LIN {X 0,Y 545.058,Z 281.586,A -85,B 0,C 180,E1 -3811.915,E2 -3811.915} C_VEL
LIN {X 0,Y 545.078,Z 281.584,A -85,B 0,C 180,E1 -3813.095,E2 -3813.095} C_VEL
LIN {X 0,Y 544.385,Z 281.672,A -85,B 0,C 180,E1 -3813.711,E2 -3813.711} C_VEL
LIN {X 0,Y 541.508,Z 282.03,A -85,B 0,C 180,E1 -3814.712,E2 -3814.712} C_VEL
LIN {X 0,Y 539.096,Z 282.331,A -85,B 0,C 180,E1 -3815.518,E2 -3815.518} C_VEL
LIN {X 0,Y 538.071,Z 282.462,A -85,B 0,C 180,E1 -3816.14,E2 -3816.14} C_VEL
LIN {X 0,Y 537.992,Z 282.467,A -85,B 0,C 180,E1 -3816.351,E2 -3816.351} C_VEL
LIN {X 0,Y 538.037,Z 282.462,A -85,B 0,C 180,E1 -3819.585,E2 -3819.585} C_VEL
LIN {X 0,Y 538.036,Z 282.468,A -85,B 0,C 180,E1 -3821.879,E2 -3821.879} C_VEL
LIN {X 0,Y 538.035,Z 282.461,A -85,B 0,C 180,E1 -3825.141,E2 -3825.141} C_VEL
LIN {X 0,Y 538.035,Z 282.463,A -85,B 0,C 180,E1 -3828.227,E2 -3828.227} C_VEL
LIN {X 0,Y 538.016,Z 282.466,A -85,B 0,C 180,E1 -3831.17,E2 -3831.17} C_VEL
LIN {X 0,Y 537.995,Z 282.469,A -85,B 0,C 180,E1 -3834.089,E2 -3834.089} C_VEL
LIN {X 0,Y 537.857,Z 282.645,A -85,B 0,C 180,E1 -3836.154,E2 -3836.154} C_VEL
LIN {X 0,Y 537.784,Z 288.557,A -85,B 0,C 180,E1 -3839.358,E2 -3839.358} C_VEL
LIN {X 0,Y 537.735,Z 293.055,A -85,B 0,C 180,E1 -3841.933,E2 -3841.933} C_VEL
LIN {X 0,Y 537.773,Z 297.369,A -85,B 0,C 180,E1 -3844.452,E2 -3844.452} C_VEL
LIN {X 0,Y 537.677,Z 301.678,A -85,B 0,C 180,E1 -3846.913,E2 -3846.913} C_VEL
LIN {X 0,Y 537.632,Z 305.956,A -85,B 0,C 180,E1 -3849.332,E2 -3849.332} C_VEL
LIN {X 0,Y 537.604,Z 310.176,A -85,B 0,C 180,E1 -3851.715,E2 -3851.715} C_VEL
LIN {X 0,Y 537.602,Z 314.303,A -85,B 0,C 180,E1 -3854.066,E2 -3854.066} C_VEL
LIN {X 0,Y 537.565,Z 318.7,A -85,B 0,C 180,E1 -3856.582,E2 -3856.582} C_VEL
LIN {X 0,Y 537.574,Z 318.943,A -85,B 0,C 180,E1 -3856.726,E2 -3856.726} C_VEL
LIN {X 0,Y 539.197,Z 329.347,A -85,B 0,C 180,E1 -3857.03,E2 -3857.03} C_VEL
LIN {X 0,Y 538.984,Z 342.462,A -85,B 0,C 180,E1 -3857.48,E2 -3857.48} C_VEL
LIN {X 0,Y 538.742,Z 354.682,A -85,B 0,C 180,E1 -3858.068,E2 -3858.068} C_VEL
LIN {X 0,Y 538.566,Z 365.025,A -85,B 0,C 180,E1 -3858.712,E2 -3858.712} C_VEL
LIN {X 0,Y 538.362,Z 374.875,A -85,B 0,C 180,E1 -3859.469,E2 -3859.469} C_VEL
LIN {X 0,Y 538.196,Z 383.038,A -85,B 0,C 180,E1 -3860.226,E2 -3860.226} C_VEL
LIN {X 0,Y 538.03,Z 389.945,A -85,B 0,C 180,E1 -3860.982,E2 -3860.982} C_VEL
LIN {X 0,Y 537.884,Z 395.929,A -85,B 0,C 180,E1 -3861.736,E2 -3861.736} C_VEL
LIN {X 0,Y 537.76,Z 402.268,A -85,B 0,C 180,E1 -3862.679,E2 -3862.679} C_VEL
LIN {X 0,Y 537.639,Z 407.848,A -85,B 0,C 180,E1 -3863.68,E2 -3863.68} C_VEL
LIN {X 0,Y 537.587,Z 412.691,A -85,B 0,C 180,E1 -3864.749,E2 -3864.749} C_VEL
LIN {X 0,Y 537.604,Z 416.69,A -85,B 0,C 180,E1 -3865.877,E2 -3865.877} C_VEL
LIN {X 0,Y 537.551,Z 419.653,A -85,B 0,C 180,E1 -3867.002,E2 -3867.002} C_VEL
LIN {X 0,Y 537.451,Z 422.149,A -85,B 0,C 180,E1 -3868.501,E2 -3868.501} C_VEL
LIN {X 0,Y 537.442,Z 422.734,A -85,B 0,C 180,E1 -3869.251,E2 -3869.251} C_VEL
LIN {X 0,Y 537.442,Z 422.804,A -85,B 0,C 180,E1 -3870.749,E2 -3870.749} C_VEL
LIN {X 0,Y 537.452,Z 422.221,A -85,B 0,C 180,E1 -3871.499,E2 -3871.499} C_VEL
LIN {X 0,Y 537.552,Z 419.867,A -85,B 0,C 180,E1 -3872.998,E2 -3872.998} C_VEL
LIN {X 0,Y 537.603,Z 416.98,A -85,B 0,C 180,E1 -3874.123,E2 -3874.123} C_VEL
LIN {X 0,Y 537.587,Z 413.06,A -85,B 0,C 180,E1 -3875.251,E2 -3875.251} C_VEL
LIN {X 0,Y 537.637,Z 408.312,A -85,B 0,C 180,E1 -3876.319,E2 -3876.319} C_VEL
LIN {X 0,Y 537.754,Z 402.817,A -85,B 0,C 180,E1 -3877.321,E2 -3877.321} C_VEL
LIN {X 0,Y 537.879,Z 396.581,A -85,B 0,C 180,E1 -3878.264,E2 -3878.264} C_VEL
LIN {X 0,Y 538.024,Z 389.105,A -85,B 0,C 180,E1 -3879.208,E2 -3879.208} C_VEL
LIN {X 0,Y 538.204,Z 382.044,A -85,B 0,C 180,E1 -3879.964,E2 -3879.964} C_VEL
LIN {X 0,Y 538.405,Z 373.693,A -85,B 0,C 180,E1 -3880.72,E2 -3880.72} C_VEL
LIN {X 0,Y 538.575,Z 363.07,A -85,B 0,C 180,E1 -3881.515,E2 -3881.515} C_VEL
LIN {X 0,Y 538.874,Z 350.602,A -85,B 0,C 180,E1 -3882.236,E2 -3882.236} C_VEL
LIN {X 0,Y 539.086,Z 338.621,A -85,B 0,C 180,E1 -3882.757,E2 -3882.757} C_VEL
LIN {X 0,Y 539.013,Z 326.997,A -85,B 0,C 180,E1 -3883.13,E2 -3883.13} C_VEL
LIN {X 0,Y 537.561,Z 318.988,A -85,B 0,C 180,E1 -3883.346,E2 -3883.346} C_VEL
LIN {X 0,Y 537.6,Z 314.46,A -85,B 0,C 180,E1 -3885.934,E2 -3885.934} C_VEL
LIN {X 0,Y 537.601,Z 310.355,A -85,B 0,C 180,E1 -3888.285,E2 -3888.285} C_VEL
LIN {X 0,Y 537.633,Z 306.122,A -85,B 0,C 180,E1 -3890.668,E2 -3890.668} C_VEL
LIN {X 0,Y 537.679,Z 301.842,A -85,B 0,C 180,E1 -3893.087,E2 -3893.087} C_VEL
LIN {X 0,Y 537.763,Z 297.422,A -85,B 0,C 180,E1 -3895.609,E2 -3895.609} C_VEL
LIN {X 0,Y 537.744,Z 291.815,A -85,B 0,C 180,E1 -3898.877,E2 -3898.877} C_VEL
LIN {X 0,Y 537.808,Z 286.54,A -85,B 0,C 180,E1 -3901.852,E2 -3901.852} C_VEL
LIN {X 0,Y 537.881,Z 282.489,A -85,B 0,C 180,E1 -3904.07,E2 -3904.07} C_VEL
LIN {X 0,Y 537.992,Z 282.474,A -85,B 0,C 180,E1 -3906.005,E2 -3906.005} C_VEL
LIN {X 0,Y 538.017,Z 282.469,A -85,B 0,C 180,E1 -3908.83,E2 -3908.83} C_VEL
LIN {X 0,Y 538.033,Z 282.466,A -85,B 0,C 180,E1 -3911.773,E2 -3911.773} C_VEL
LIN {X 0,Y 538.008,Z 282.472,A -85,B 0,C 180,E1 -3914.862,E2 -3914.862} C_VEL
LIN {X 0,Y 538.022,Z 282.468,A -85,B 0,C 180,E1 -3917.214,E2 -3917.214} C_VEL
LIN {X 0,Y 538.029,Z 282.47,A -85,B 0,C 180,E1 -3920.203,E2 -3920.203} C_VEL
LIN {X 0,Y 538.022,Z 282.468,A -85,B 0,C 180,E1 -3923.067,E2 -3923.067} C_VEL
LIN {X 0,Y 537.896,Z 282.486,A -85,B 0,C 180,E1 -3926.044,E2 -3926.044} C_VEL
LIN {X 0,Y 537.837,Z 282.622,A -85,B 0,C 180,E1 -3926.265,E2 -3926.265} C_VEL
LIN {X 0,Y 537.782,Z 288.721,A -85,B 0,C 180,E1 -3929.601,E2 -3929.601} C_VEL
LIN {X 0,Y 537.749,Z 294.411,A -85,B 0,C 180,E1 -3932.779,E2 -3932.779} C_VEL
LIN {X 0,Y 537.75,Z 298.878,A -85,B 0,C 180,E1 -3935.278,E2 -3935.278} C_VEL
LIN {X 0,Y 537.696,Z 304.615,A -85,B 0,C 180,E1 -3938.532,E2 -3938.532} C_VEL
LIN {X 0,Y 537.649,Z 308.817,A -85,B 0,C 180,E1 -3940.926,E2 -3940.926} C_VEL
LIN {X 0,Y 537.608,Z 313.006,A -85,B 0,C 180,E1 -3943.286,E2 -3943.286} C_VEL
LIN {X 0,Y 537.616,Z 316.936,A -85,B 0,C 180,E1 -3945.618,E2 -3945.618} C_VEL
LIN {X 0,Y 537.549,Z 318.912,A -85,B 0,C 180,E1 -3946.762,E2 -3946.762} C_VEL
LIN {X 0,Y 539.18,Z 328.814,A -85,B 0,C 180,E1 -3947.03,E2 -3947.03} C_VEL
LIN {X 0,Y 539.005,Z 342.142,A -85,B 0,C 180,E1 -3947.48,E2 -3947.48} C_VEL
LIN {X 0,Y 538.747,Z 353.631,A -85,B 0,C 180,E1 -3948.028,E2 -3948.028} C_VEL
LIN {X 0,Y 538.577,Z 363.06,A -85,B 0,C 180,E1 -3948.592,E2 -3948.592} C_VEL
LIN {X 0,Y 538.43,Z 371.298,A -85,B 0,C 180,E1 -3949.185,E2 -3949.185} C_VEL
LIN {X 0,Y 538.233,Z 379.087,A -85,B 0,C 180,E1 -3949.847,E2 -3949.847} C_VEL
LIN {X 0,Y 538.077,Z 386.623,A -85,B 0,C 180,E1 -3950.603,E2 -3950.603} C_VEL
LIN {X 0,Y 537.974,Z 393.094,A -85,B 0,C 180,E1 -3951.359,E2 -3951.359} C_VEL
LIN {X 0,Y 537.82,Z 399.898,A -85,B 0,C 180,E1 -3952.302,E2 -3952.302} C_VEL
LIN {X 0,Y 537.718,Z 405.583,A -85,B 0,C 180,E1 -3953.245,E2 -3953.245} C_VEL
LIN {X 0,Y 537.675,Z 411.113,A -85,B 0,C 180,E1 -3954.374,E2 -3954.374} C_VEL
LIN {X 0,Y 537.562,Z 415.464,A -85,B 0,C 180,E1 -3955.501,E2 -3955.501} C_VEL
LIN {X 0,Y 537.591,Z 417.825,A -85,B 0,C 180,E1 -3956.252,E2 -3956.252} C_VEL
LIN {X 0,Y 537.551,Z 419.682,A -85,B 0,C 180,E1 -3957.002,E2 -3957.002} C_VEL
LIN {X 0,Y 537.451,Z 422.122,A -85,B 0,C 180,E1 -3958.501,E2 -3958.501} C_VEL
LIN {X 0,Y 537.442,Z 422.755,A -85,B 0,C 180,E1 -3959.251,E2 -3959.251} C_VEL
LIN {X 0,Y 537.442,Z 422.786,A -85,B 0,C 180,E1 -3960.749,E2 -3960.749} C_VEL
LIN {X 0,Y 537.452,Z 422.232,A -85,B 0,C 180,E1 -3961.499,E2 -3961.499} C_VEL
LIN {X 0,Y 537.552,Z 419.859,A -85,B 0,C 180,E1 -3962.998,E2 -3962.998} C_VEL
LIN {X 0,Y 537.603,Z 416.977,A -85,B 0,C 180,E1 -3964.123,E2 -3964.123} C_VEL
LIN {X 0,Y 537.587,Z 413.06,A -85,B 0,C 180,E1 -3965.251,E2 -3965.251} C_VEL
LIN {X 0,Y 537.639,Z 408.305,A -85,B 0,C 180,E1 -3966.32,E2 -3966.32} C_VEL
LIN {X 0,Y 537.754,Z 402.819,A -85,B 0,C 180,E1 -3967.321,E2 -3967.321} C_VEL
LIN {X 0,Y 537.875,Z 396.582,A -85,B 0,C 180,E1 -3968.264,E2 -3968.264} C_VEL
LIN {X 0,Y 537.982,Z 390.729,A -85,B 0,C 180,E1 -3969.019,E2 -3969.019} C_VEL
LIN {X 0,Y 538.134,Z 383.935,A -85,B 0,C 180,E1 -3969.775,E2 -3969.775} C_VEL
LIN {X 0,Y 538.368,Z 374.742,A -85,B 0,C 180,E1 -3970.626,E2 -3970.626} C_VEL
LIN {X 0,Y 538.509,Z 366.147,A -85,B 0,C 180,E1 -3971.289,E2 -3971.289} C_VEL
LIN {X 0,Y 538.674,Z 356.599,A -85,B 0,C 180,E1 -3971.897,E2 -3971.897} C_VEL
LIN {X 0,Y 538.872,Z 346.258,A -85,B 0,C 180,E1 -3972.427,E2 -3972.427} C_VEL
LIN {X 0,Y 539.084,Z 335.494,A -85,B 0,C 180,E1 -3972.853,E2 -3972.853} C_VEL
LIN {X 0,Y 538.998,Z 327.101,A -85,B 0,C 180,E1 -3973.106,E2 -3973.106} C_VEL
LIN {X 0,Y 537.553,Z 319.061,A -85,B 0,C 180,E1 -3973.322,E2 -3973.322} C_VEL
LIN {X 0,Y 537.613,Z 314.728,A -85,B 0,C 180,E1 -3975.934,E2 -3975.934} C_VEL
LIN {X 0,Y 537.661,Z 309.18,A -85,B 0,C 180,E1 -3979.074,E2 -3979.074} C_VEL
LIN {X 0,Y 537.727,Z 304.116,A -85,B 0,C 180,E1 -3981.881,E2 -3981.881} C_VEL
LIN {X 0,Y 537.695,Z 298.715,A -85,B 0,C 180,E1 -3984.725,E2 -3984.725} C_VEL
LIN {X 0,Y 537.669,Z 293.664,A -85,B 0,C 180,E1 -3987.271,E2 -3987.271} C_VEL
LIN {X 0,Y 537.56,Z 288.115,A -85,B 0,C 180,E1 -3989.789,E2 -3989.789} C_VEL
LIN {X 0,Y 537.606,Z 282.523,A -85,B 0,C 180,E1 -3992.165,E2 -3992.165} C_VEL
LIN {X 0,Y 537.962,Z 282.477,A -85,B 0,C 180,E1 -3994.178,E2 -3994.178} C_VEL
LIN {X 0,Y 538.005,Z 282.47,A -85,B 0,C 180,E1 -3997.17,E2 -3997.17} C_VEL
LIN {X 0,Y 538.024,Z 282.467,A -85,B 0,C 180,E1 -3999.797,E2 -3999.797} C_VEL
LIN {X 0,Y 538.002,Z 282.471,A -85,B 0,C 180,E1 -4002.788,E2 -4002.788} C_VEL
LIN {X 0,Y 538.035,Z 282.466,A -85,B 0,C 180,E1 -4005.141,E2 -4005.141} C_VEL
LIN {X 0,Y 538.025,Z 282.469,A -85,B 0,C 180,E1 -4008.226,E2 -4008.226} C_VEL
LIN {X 0,Y 538.014,Z 282.472,A -85,B 0,C 180,E1 -4011.169,E2 -4011.169} C_VEL
LIN {X 0,Y 538.02,Z 282.572,A -85,B 0,C 180,E1 -4011.607,E2 -4011.607} C_VEL
LIN {X 0,Y 539.515,Z 290.583,A -85,B 0,C 180,E1 -4014.113,E2 -4014.113} C_VEL
LIN {X 0,Y 539.286,Z 299.975,A -85,B 0,C 180,E1 -4016.815,E2 -4016.815} C_VEL
LIN {X 0,Y 539.077,Z 309.293,A -85,B 0,C 180,E1 -4019.439,E2 -4019.439} C_VEL
LIN {X 0,Y 538.798,Z 320.333,A -85,B 0,C 180,E1 -4022.497,E2 -4022.497} C_VEL
LIN {X 0,Y 538.543,Z 330.78,A -85,B 0,C 180,E1 -4025.317,E2 -4025.317} C_VEL
LIN {X 0,Y 538.364,Z 340.735,A -85,B 0,C 180,E1 -4027.951,E2 -4027.951} C_VEL
LIN {X 0,Y 538.15,Z 352.266,A -85,B 0,C 180,E1 -4030.944,E2 -4030.944} C_VEL
LIN {X 0,Y 537.953,Z 363.009,A -85,B 0,C 180,E1 -4033.687,E2 -4033.687} C_VEL
LIN {X 0,Y 537.827,Z 374.712,A -85,B 0,C 180,E1 -4036.636,E2 -4036.636} C_VEL
LIN {X 0,Y 539.239,Z 384.519,A -85,B 0,C 180,E1 -4036.864,E2 -4036.864} C_VEL
LIN {X 0,Y 539.091,Z 397.175,A -85,B 0,C 180,E1 -4037.243,E2 -4037.243} C_VEL
LIN {X 0,Y 538.845,Z 409.485,A -85,B 0,C 180,E1 -4037.764,E2 -4037.764} C_VEL
LIN {X 0,Y 538.65,Z 420.458,A -85,B 0,C 180,E1 -4038.374,E2 -4038.374} C_VEL
LIN {X 0,Y 538.413,Z 431.925,A -85,B 0,C 180,E1 -4039.185,E2 -4039.185} C_VEL
LIN {X 0,Y 538.2,Z 441.6,A -85,B 0,C 180,E1 -4040.036,E2 -4040.036} C_VEL
LIN {X 0,Y 538.015,Z 450.412,A -85,B 0,C 180,E1 -4040.981,E2 -4040.981} C_VEL
LIN {X 0,Y 537.829,Z 459.001,A -85,B 0,C 180,E1 -4042.114,E2 -4042.114} C_VEL
LIN {X 0,Y 537.705,Z 465.868,A -85,B 0,C 180,E1 -4043.244,E2 -4043.244} C_VEL
LIN {X 0,Y 537.676,Z 471.366,A -85,B 0,C 180,E1 -4044.374,E2 -4044.374} C_VEL
LIN {X 0,Y 537.557,Z 475.677,A -85,B 0,C 180,E1 -4045.501,E2 -4045.501} C_VEL
LIN {X 0,Y 537.591,Z 477.957,A -85,B 0,C 180,E1 -4046.252,E2 -4046.252} C_VEL
LIN {X 0,Y 537.551,Z 479.808,A -85,B 0,C 180,E1 -4047.002,E2 -4047.002} C_VEL
LIN {X 0,Y 537.49,Z 481.198,A -85,B 0,C 180,E1 -4047.752,E2 -4047.752} C_VEL
LIN {X 0,Y 537.442,Z 482.785,A -85,B 0,C 180,E1 -4049.251,E2 -4049.251} C_VEL
LIN {X 0,Y 537.442,Z 483,A -85,B 0,C 180,E1 -4050,E2 -4050} C_VEL
LIN {X 0,Y 537.451,Z 482.186,A -85,B 0,C 180,E1 -4051.499,E2 -4051.499} C_VEL
LIN {X 0,Y 537.49,Z 481.199,A -85,B 0,C 180,E1 -4052.248,E2 -4052.248} C_VEL
LIN {X 0,Y 537.551,Z 479.81,A -85,B 0,C 180,E1 -4052.998,E2 -4052.998} C_VEL
LIN {X 0,Y 537.603,Z 476.896,A -85,B 0,C 180,E1 -4054.123,E2 -4054.123} C_VEL
LIN {X 0,Y 537.587,Z 472.949,A -85,B 0,C 180,E1 -4055.251,E2 -4055.251} C_VEL
LIN {X 0,Y 537.652,Z 468.087,A -85,B 0,C 180,E1 -4056.334,E2 -4056.334} C_VEL
LIN {X 0,Y 537.791,Z 461.468,A -85,B 0,C 180,E1 -4057.509,E2 -4057.509} C_VEL
LIN {X 0,Y 537.972,Z 453.478,A -85,B 0,C 180,E1 -4058.641,E2 -4058.641} C_VEL
LIN {X 0,Y 538.119,Z 445.335,A -85,B 0,C 180,E1 -4059.586,E2 -4059.586} C_VEL
LIN {X 0,Y 538.375,Z 435.4,A -85,B 0,C 180,E1 -4060.53,E2 -4060.53} C_VEL
LIN {X 0,Y 538.542,Z 425.586,A -85,B 0,C 180,E1 -4061.289,E2 -4061.289} C_VEL
LIN {X 0,Y 538.74,Z 414.594,A -85,B 0,C 180,E1 -4061.971,E2 -4061.971} C_VEL
LIN {X 0,Y 538.94,Z 402.108,A -85,B 0,C 180,E1 -4062.569,E2 -4062.569} C_VEL
LIN {X 0,Y 539.197,Z 389.087,A -85,B 0,C 180,E1 -4063.017,E2 -4063.017} C_VEL
LIN {X 0,Y 539.058,Z 382.364,A -85,B 0,C 180,E1 -4063.189,E2 -4063.189} C_VEL
LIN {X 0,Y 537.827,Z 374.712,A -85,B 0,C 180,E1 -4063.364,E2 -4063.364} C_VEL
LIN {X 0,Y 537.953,Z 363.009,A -85,B 0,C 180,E1 -4066.313,E2 -4066.313} C_VEL
LIN {X 0,Y 538.15,Z 352.266,A -85,B 0,C 180,E1 -4069.056,E2 -4069.056} C_VEL
LIN {X 0,Y 538.398,Z 339.988,A -85,B 0,C 180,E1 -4072.244,E2 -4072.244} C_VEL
LIN {X 0,Y 538.543,Z 330.78,A -85,B 0,C 180,E1 -4074.683,E2 -4074.683} C_VEL
LIN {X 0,Y 538.798,Z 320.333,A -85,B 0,C 180,E1 -4077.503,E2 -4077.503} C_VEL
LIN {X 0,Y 539.091,Z 309.026,A -85,B 0,C 180,E1 -4080.635,E2 -4080.635} C_VEL
LIN {X 0,Y 539.219,Z 299.631,A -85,B 0,C 180,E1 -4083.19,E2 -4083.19} C_VEL
LIN {X 0,Y 539.368,Z 291.385,A -85,B 0,C 180,E1 -4085.439,E2 -4085.439} C_VEL
LIN {X 0,Y 538.769,Z 286.486,A -85,B 0,C 180,E1 -4086.874,E2 -4086.874} C_VEL
LIN {X 0,Y 538.029,Z 282.469,A -85,B 0,C 180,E1 -4088.199,E2 -4088.199} C_VEL
LIN {X 0,Y 538.004,Z 282.473,A -85,B 0,C 180,E1 -4090.78,E2 -4090.78} C_VEL
LIN {X 0,Y 538.013,Z 282.468,A -85,B 0,C 180,E1 -4094.072,E2 -4094.072} C_VEL
LIN {X 0,Y 538,Z 282.469,A -85,B 0,C 180,E1 -4097.016,E2 -4097.016} C_VEL
LIN {X 0,Y 538.051,Z 282.461,A -85,B 0,C 180,E1 -4099.253,E2 -4099.253} C_VEL
LIN {X 0,Y 537.995,Z 282.474,A -85,B 0,C 180,E1 -4102.122,E2 -4102.122} C_VEL
LIN {X 0,Y 538.001,Z 282.467,A -85,B 0,C 180,E1 -4104.916,E2 -4104.916} C_VEL
LIN {X 0,Y 538.022,Z 282.47,A -85,B 0,C 180,E1 -4107.617,E2 -4107.617} C_VEL
LIN {X 0,Y 538.02,Z 282.467,A -85,B 0,C 180,E1 -4110.239,E2 -4110.239} C_VEL
LIN {X 0,Y 538.061,Z 282.461,A -85,B 0,C 180,E1 -4112.796,E2 -4112.796} C_VEL
LIN {X 0,Y 537.956,Z 282.479,A -85,B 0,C 180,E1 -4115.288,E2 -4115.288} C_VEL
LIN {X 0,Y 537.83,Z 282.494,A -85,B 0,C 180,E1 -4116.92,E2 -4116.92} C_VEL
LIN {X 0,Y 537.786,Z 283.612,A -85,B 0,C 180,E1 -4118.536,E2 -4118.536} C_VEL
LIN {X 0,Y 537.704,Z 285.905,A -85,B 0,C 180,E1 -4120.928,E2 -4120.928} C_VEL
LIN {X 0,Y 537.624,Z 287.92,A -85,B 0,C 180,E1 -4123.286,E2 -4123.286} C_VEL
LIN {X 0,Y 537.615,Z 289.979,A -85,B 0,C 180,E1 -4125.618,E2 -4125.618} C_VEL
LIN {X 0,Y 537.573,Z 291.236,A -85,B 0,C 180,E1 -4126.798,E2 -4126.798} C_VEL
LIN {X 0,Y 539.171,Z 300.777,A -85,B 0,C 180,E1 -4127.078,E2 -4127.078} C_VEL
LIN {X 0,Y 538.979,Z 312.274,A -85,B 0,C 180,E1 -4127.48,E2 -4127.48} C_VEL
LIN {X 0,Y 538.774,Z 322.521,A -85,B 0,C 180,E1 -4127.953,E2 -4127.953} C_VEL
LIN {X 0,Y 538.649,Z 331.507,A -85,B 0,C 180,E1 -4128.472,E2 -4128.472} C_VEL
LIN {X 0,Y 538.45,Z 340.354,A -85,B 0,C 180,E1 -4129.091,E2 -4129.091} C_VEL
LIN {X 0,Y 538.292,Z 348.295,A -85,B 0,C 180,E1 -4129.753,E2 -4129.753} C_VEL
LIN {X 0,Y 538.143,Z 355.087,A -85,B 0,C 180,E1 -4130.415,E2 -4130.415} C_VEL
LIN {X 0,Y 537.981,Z 361.742,A -85,B 0,C 180,E1 -4131.17,E2 -4131.17} C_VEL
LIN {X 0,Y 537.832,Z 368.713,A -85,B 0,C 180,E1 -4132.114,E2 -4132.114} C_VEL
LIN {X 0,Y 537.74,Z 374.517,A -85,B 0,C 180,E1 -4133.056,E2 -4133.056} C_VEL
LIN {X 0,Y 537.695,Z 379.406,A -85,B 0,C 180,E1 -4133.998,E2 -4133.998} C_VEL
LIN {X 0,Y 537.54,Z 384.136,A -85,B 0,C 180,E1 -4135.125,E2 -4135.125} C_VEL
LIN {X 0,Y 537.591,Z 387.77,A -85,B 0,C 180,E1 -4136.252,E2 -4136.252} C_VEL
LIN {X 0,Y 537.551,Z 389.661,A -85,B 0,C 180,E1 -4137.002,E2 -4137.002} C_VEL
LIN {X 0,Y 537.49,Z 391.132,A -85,B 0,C 180,E1 -4137.752,E2 -4137.752} C_VEL
LIN {X 0,Y 537.442,Z 392.717,A -85,B 0,C 180,E1 -4139.251,E2 -4139.251} C_VEL
LIN {X 0,Y 537.442,Z 392.996,A -85,B 0,C 180,E1 -4140,E2 -4140} C_VEL
LIN {X 0,Y 537.452,Z 392.187,A -85,B 0,C 180,E1 -4141.499,E2 -4141.499} C_VEL
LIN {X 0,Y 537.49,Z 391.282,A -85,B 0,C 180,E1 -4142.248,E2 -4142.248} C_VEL
LIN {X 0,Y 537.591,Z 388.019,A -85,B 0,C 180,E1 -4143.748,E2 -4143.748} C_VEL
LIN {X 0,Y 537.54,Z 384.465,A -85,B 0,C 180,E1 -4144.875,E2 -4144.875} C_VEL
LIN {X 0,Y 537.668,Z 379.815,A -85,B 0,C 180,E1 -4146.002,E2 -4146.002} C_VEL
LIN {X 0,Y 537.729,Z 373.953,A -85,B 0,C 180,E1 -4147.132,E2 -4147.132} C_VEL
LIN {X 0,Y 537.871,Z 366.768,A -85,B 0,C 180,E1 -4148.264,E2 -4148.264} C_VEL
LIN {X 0,Y 538.053,Z 357.614,A -85,B 0,C 180,E1 -4149.397,E2 -4149.397} C_VEL
LIN {X 0,Y 538.254,Z 349.208,A -85,B 0,C 180,E1 -4150.248,E2 -4150.248} C_VEL
LIN {X 0,Y 538.462,Z 340.199,A -85,B 0,C 180,E1 -4151.005,E2 -4151.005} C_VEL
LIN {X 0,Y 538.647,Z 330.368,A -85,B 0,C 180,E1 -4151.684,E2 -4151.684} C_VEL
LIN {X 0,Y 538.836,Z 320.495,A -85,B 0,C 180,E1 -4152.237,E2 -4152.237} C_VEL
LIN {X 0,Y 539.066,Z 308.575,A -85,B 0,C 180,E1 -4152.757,E2 -4152.757} C_VEL
LIN {X 0,Y 538.999,Z 298.562,A -85,B 0,C 180,E1 -4153.082,E2 -4153.082} C_VEL
LIN {X 0,Y 537.539,Z 290.625,A -85,B 0,C 180,E1 -4153.323,E2 -4153.323} C_VEL
LIN {X 0,Y 537.527,Z 287.909,A -85,B 0,C 180,E1 -4155.936,E2 -4155.936} C_VEL
LIN {X 0,Y 537.529,Z 285.425,A -85,B 0,C 180,E1 -4158.288,E2 -4158.288} C_VEL
LIN {X 0,Y 537.557,Z 282.839,A -85,B 0,C 180,E1 -4160.671,E2 -4160.671} C_VEL
LIN {X 0,Y 537.728,Z 282.507,A -85,B 0,C 180,E1 -4162.273,E2 -4162.273} C_VEL
LIN {X 0,Y 537.946,Z 282.48,A -85,B 0,C 180,E1 -4164.713,E2 -4164.713} C_VEL
LIN {X 0,Y 538.051,Z 282.458,A -85,B 0,C 180,E1 -4167.35,E2 -4167.35} C_VEL
LIN {X 0,Y 538.018,Z 282.463,A -85,B 0,C 180,E1 -4169.761,E2 -4169.761} C_VEL
LIN {X 0,Y 538.021,Z 282.469,A -85,B 0,C 180,E1 -4172.383,E2 -4172.383} C_VEL
LIN {X 0,Y 538.001,Z 282.464,A -85,B 0,C 180,E1 -4175.084,E2 -4175.084} C_VEL
LIN {X 0,Y 537.992,Z 282.467,A -85,B 0,C 180,E1 -4176.351,E2 -4176.351} C_VEL
LIN {X 0,Y 537.342,Z 282.55,A -85,B 0,C 180,E1 -4176.976,E2 -4176.976} C_VEL
LIN {X 0,Y 534.507,Z 282.907,A -85,B 0,C 180,E1 -4177.991,E2 -4177.991} C_VEL
LIN {X 0,Y 532.101,Z 283.202,A -85,B 0,C 180,E1 -4178.809,E2 -4178.809} C_VEL
LIN {X 0,Y 531.067,Z 283.33,A -85,B 0,C 180,E1 -4179.44,E2 -4179.44} C_VEL
LIN {X 0,Y 530.982,Z 283.342,A -85,B 0,C 180,E1 -4179.653,E2 -4179.653} C_VEL
LIN {X 0,Y 530.983,Z 283.343,A -85,B 0,C 180,E1 -4182.457,E2 -4182.457} C_VEL
LIN {X 0,Y 530.992,Z 283.343,A -85,B 0,C 180,E1 -4185.621,E2 -4185.621} C_VEL
LIN {X 0,Y 530.998,Z 283.338,A -85,B 0,C 180,E1 -4188.565,E2 -4188.565} C_VEL
LIN {X 0,Y 530.961,Z 283.349,A -85,B 0,C 180,E1 -4191.529,E2 -4191.529} C_VEL
LIN {X 0,Y 530.947,Z 283.346,A -85,B 0,C 180,E1 -4194.379,E2 -4194.379} C_VEL
LIN {X 0,Y 530.792,Z 283.494,A -85,B 0,C 180,E1 -4196.213,E2 -4196.213} C_VEL
LIN {X 0,Y 530.742,Z 288.452,A -85,B 0,C 180,E1 -4198.907,E2 -4198.907} C_VEL
LIN {X 0,Y 530.658,Z 293.031,A -85,B 0,C 180,E1 -4201.524,E2 -4201.524} C_VEL
LIN {X 0,Y 530.68,Z 297.632,A -85,B 0,C 180,E1 -4204.231,E2 -4204.231} C_VEL
LIN {X 0,Y 530.635,Z 301.709,A -85,B 0,C 180,E1 -4206.588,E2 -4206.588} C_VEL
LIN {X 0,Y 530.58,Z 306.024,A -85,B 0,C 180,E1 -4209.045,E2 -4209.045} C_VEL
LIN {X 0,Y 530.534,Z 310.312,A -85,B 0,C 180,E1 -4211.462,E2 -4211.462} C_VEL
LIN {X 0,Y 530.536,Z 314.532,A -85,B 0,C 180,E1 -4213.848,E2 -4213.848} C_VEL
LIN {X 0,Y 530.511,Z 319.204,A -85,B 0,C 180,E1 -4216.497,E2 -4216.497} C_VEL
LIN {X 0,Y 530.544,Z 319.671,A -85,B 0,C 180,E1 -4216.571,E2 -4216.571} C_VEL
LIN {X 0,Y 532.299,Z 329.735,A -85,B 0,C 180,E1 -4216.859,E2 -4216.859} C_VEL
LIN {X 0,Y 532.086,Z 342.841,A -85,B 0,C 180,E1 -4217.315,E2 -4217.315} C_VEL
LIN {X 0,Y 531.854,Z 354.465,A -85,B 0,C 180,E1 -4217.876,E2 -4217.876} C_VEL
LIN {X 0,Y 531.624,Z 365.46,A -85,B 0,C 180,E1 -4218.562,E2 -4218.562} C_VEL
LIN {X 0,Y 531.394,Z 376.467,A -85,B 0,C 180,E1 -4219.426,E2 -4219.426} C_VEL
LIN {X 0,Y 531.168,Z 385.371,A -85,B 0,C 180,E1 -4220.288,E2 -4220.288} C_VEL
LIN {X 0,Y 530.921,Z 394.959,A -85,B 0,C 180,E1 -4221.436,E2 -4221.436} C_VEL
LIN {X 0,Y 530.723,Z 402.633,A -85,B 0,C 180,E1 -4222.582,E2 -4222.582} C_VEL
LIN {X 0,Y 530.598,Z 408.624,A -85,B 0,C 180,E1 -4223.694,E2 -4223.694} C_VEL
LIN {X 0,Y 530.523,Z 412.913,A -85,B 0,C 180,E1 -4224.679,E2 -4224.679} C_VEL
LIN {X 0,Y 530.524,Z 416.848,A -85,B 0,C 180,E1 -4225.822,E2 -4225.822} C_VEL
LIN {X 0,Y 530.457,Z 419.771,A -85,B 0,C 180,E1 -4226.962,E2 -4226.962} C_VEL
LIN {X 0,Y 530.361,Z 422.226,A -85,B 0,C 180,E1 -4228.481,E2 -4228.481} C_VEL
LIN {X 0,Y 530.344,Z 422.815,A -85,B 0,C 180,E1 -4229.241,E2 -4229.241} C_VEL
LIN {X 0,Y 530.344,Z 422.874,A -85,B 0,C 180,E1 -4230.759,E2 -4230.759} C_VEL
LIN {X 0,Y 530.362,Z 422.308,A -85,B 0,C 180,E1 -4231.519,E2 -4231.519} C_VEL
LIN {X 0,Y 530.457,Z 419.975,A -85,B 0,C 180,E1 -4233.038,E2 -4233.038} C_VEL
LIN {X 0,Y 530.522,Z 417.13,A -85,B 0,C 180,E1 -4234.178,E2 -4234.178} C_VEL
LIN {X 0,Y 530.524,Z 413.272,A -85,B 0,C 180,E1 -4235.321,E2 -4235.321} C_VEL
LIN {X 0,Y 530.622,Z 407.604,A -85,B 0,C 180,E1 -4236.603,E2 -4236.603} C_VEL
LIN {X 0,Y 530.779,Z 400.832,A -85,B 0,C 180,E1 -4237.8,E2 -4237.8} C_VEL
LIN {X 0,Y 530.965,Z 392.736,A -85,B 0,C 180,E1 -4238.947,E2 -4238.947} C_VEL
LIN {X 0,Y 531.159,Z 384.396,A -85,B 0,C 180,E1 -4239.905,E2 -4239.905} C_VEL
LIN {X 0,Y 531.431,Z 374.14,A -85,B 0,C 180,E1 -4240.862,E2 -4240.862} C_VEL
LIN {X 0,Y 531.633,Z 363.877,A -85,B 0,C 180,E1 -4241.639,E2 -4241.639} C_VEL
LIN {X 0,Y 531.9,Z 352.842,A -85,B 0,C 180,E1 -4242.302,E2 -4242.302} C_VEL
LIN {X 0,Y 532.139,Z 340.239,A -85,B 0,C 180,E1 -4242.878,E2 -4242.878} C_VEL
LIN {X 0,Y 532.189,Z 328.249,A -85,B 0,C 180,E1 -4243.277,E2 -4243.277} C_VEL
LIN {X 0,Y 530.518,Z 319.32,A -85,B 0,C 180,E1 -4243.527,E2 -4243.527} C_VEL
LIN {X 0,Y 530.535,Z 314.703,A -85,B 0,C 180,E1 -4246.152,E2 -4246.152} C_VEL
LIN {X 0,Y 530.533,Z 310.484,A -85,B 0,C 180,E1 -4248.538,E2 -4248.538} C_VEL
LIN {X 0,Y 530.58,Z 306.191,A -85,B 0,C 180,E1 -4250.955,E2 -4250.955} C_VEL
LIN {X 0,Y 530.672,Z 300.899,A -85,B 0,C 180,E1 -4253.962,E2 -4253.962} C_VEL
LIN {X 0,Y 530.64,Z 296.104,A -85,B 0,C 180,E1 -4256.764,E2 -4256.764} C_VEL
LIN {X 0,Y 530.667,Z 291.696,A -85,B 0,C 180,E1 -4259.342,E2 -4259.342} C_VEL
LIN {X 0,Y 530.752,Z 286.867,A -85,B 0,C 180,E1 -4262.063,E2 -4262.063} C_VEL
LIN {X 0,Y 530.807,Z 283.37,A -85,B 0,C 180,E1 -4264.014,E2 -4264.014} C_VEL
LIN {X 0,Y 530.942,Z 283.351,A -85,B 0,C 180,E1 -4266.152,E2 -4266.152} C_VEL
LIN {X 0,Y 530.97,Z 283.348,A -85,B 0,C 180,E1 -4268.654,E2 -4268.654} C_VEL
LIN {X 0,Y 530.996,Z 283.343,A -85,B 0,C 180,E1 -4271.436,E2 -4271.436} C_VEL
LIN {X 0,Y 530.976,Z 283.346,A -85,B 0,C 180,E1 -4274.548,E2 -4274.548} C_VEL
LIN {X 0,Y 530.985,Z 283.345,A -85,B 0,C 180,E1 -4277.834,E2 -4277.834} C_VEL
LIN {X 0,Y 530.991,Z 283.343,A -85,B 0,C 180,E1 -4280.557,E2 -4280.557} C_VEL
LIN {X 0,Y 530.953,Z 283.348,A -85,B 0,C 180,E1 -4283.441,E2 -4283.441} C_VEL
LIN {X 0,Y 530.928,Z 283.352,A -85,B 0,C 180,E1 -4285.305,E2 -4285.305} C_VEL
LIN {X 0,Y 530.772,Z 283.442,A -85,B 0,C 180,E1 -4286.308,E2 -4286.308} C_VEL
LIN {X 0,Y 530.709,Z 289.065,A -85,B 0,C 180,E1 -4289.404,E2 -4289.404} C_VEL
LIN {X 0,Y 530.66,Z 294.691,A -85,B 0,C 180,E1 -4292.541,E2 -4292.541} C_VEL
LIN {X 0,Y 530.677,Z 298.921,A -85,B 0,C 180,E1 -4294.926,E2 -4294.926} C_VEL
LIN {X 0,Y 530.606,Z 304.337,A -85,B 0,C 180,E1 -4297.998,E2 -4297.998} C_VEL
LIN {X 0,Y 530.587,Z 308.987,A -85,B 0,C 180,E1 -4300.662,E2 -4300.662} C_VEL
LIN {X 0,Y 530.554,Z 313.208,A -85,B 0,C 180,E1 -4303.057,E2 -4303.057} C_VEL
LIN {X 0,Y 530.576,Z 317.205,A -85,B 0,C 180,E1 -4305.423,E2 -4305.423} C_VEL
LIN {X 0,Y 530.486,Z 319.187,A -85,B 0,C 180,E1 -4306.594,E2 -4306.594} C_VEL
LIN {X 0,Y 532.236,Z 329.509,A -85,B 0,C 180,E1 -4306.882,E2 -4306.882} C_VEL
LIN {X 0,Y 532.031,Z 343.207,A -85,B 0,C 180,E1 -4307.362,E2 -4307.362} C_VEL
LIN {X 0,Y 531.781,Z 354.258,A -85,B 0,C 180,E1 -4307.9,E2 -4307.9} C_VEL
LIN {X 0,Y 531.604,Z 363.383,A -85,B 0,C 180,E1 -4308.454,E2 -4308.454} C_VEL
LIN {X 0,Y 531.415,Z 372.652,A -85,B 0,C 180,E1 -4309.137,E2 -4309.137} C_VEL
LIN {X 0,Y 531.2,Z 381.287,A -85,B 0,C 180,E1 -4309.904,E2 -4309.904} C_VEL
LIN {X 0,Y 531.046,Z 388.551,A -85,B 0,C 180,E1 -4310.67,E2 -4310.67} C_VEL
LIN {X 0,Y 530.888,Z 394.76,A -85,B 0,C 180,E1 -4311.435,E2 -4311.435} C_VEL
LIN {X 0,Y 530.767,Z 401.315,A -85,B 0,C 180,E1 -4312.391,E2 -4312.391} C_VEL
LIN {X 0,Y 530.671,Z 405.796,A -85,B 0,C 180,E1 -4313.154,E2 -4313.154} C_VEL
LIN {X 0,Y 530.609,Z 411.288,A -85,B 0,C 180,E1 -4314.299,E2 -4314.299} C_VEL
LIN {X 0,Y 530.468,Z 415.607,A -85,B 0,C 180,E1 -4315.441,E2 -4315.441} C_VEL
LIN {X 0,Y 530.516,Z 417.944,A -85,B 0,C 180,E1 -4316.202,E2 -4316.202} C_VEL
LIN {X 0,Y 530.457,Z 419.779,A -85,B 0,C 180,E1 -4316.962,E2 -4316.962} C_VEL
LIN {X 0,Y 530.361,Z 422.199,A -85,B 0,C 180,E1 -4318.481,E2 -4318.481} C_VEL
LIN {X 0,Y 530.344,Z 422.824,A -85,B 0,C 180,E1 -4319.241,E2 -4319.241} C_VEL
LIN {X 0,Y 530.344,Z 422.858,A -85,B 0,C 180,E1 -4320.759,E2 -4320.759} C_VEL
LIN {X 0,Y 530.362,Z 422.311,A -85,B 0,C 180,E1 -4321.519,E2 -4321.519} C_VEL
LIN {X 0,Y 530.457,Z 419.964,A -85,B 0,C 180,E1 -4323.038,E2 -4323.038} C_VEL
LIN {X 0,Y 530.522,Z 417.112,A -85,B 0,C 180,E1 -4324.178,E2 -4324.178} C_VEL
LIN {X 0,Y 530.524,Z 413.239,A -85,B 0,C 180,E1 -4325.321,E2 -4325.321} C_VEL
LIN {X 0,Y 530.575,Z 409.017,A -85,B 0,C 180,E1 -4326.306,E2 -4326.306} C_VEL
LIN {X 0,Y 530.712,Z 403.076,A -85,B 0,C 180,E1 -4327.418,E2 -4327.418} C_VEL
LIN {X 0,Y 530.839,Z 396.869,A -85,B 0,C 180,E1 -4328.374,E2 -4328.374} C_VEL
LIN {X 0,Y 531.021,Z 389.388,A -85,B 0,C 180,E1 -4329.33,E2 -4329.33} C_VEL
LIN {X 0,Y 531.21,Z 382.258,A -85,B 0,C 180,E1 -4330.096,E2 -4330.096} C_VEL
LIN {X 0,Y 531.386,Z 373.801,A -85,B 0,C 180,E1 -4330.863,E2 -4330.863} C_VEL
LIN {X 0,Y 531.585,Z 364.802,A -85,B 0,C 180,E1 -4331.543,E2 -4331.543} C_VEL
LIN {X 0,Y 531.745,Z 355.836,A -85,B 0,C 180,E1 -4332.103,E2 -4332.103} C_VEL
LIN {X 0,Y 531.99,Z 344.14,A -85,B 0,C 180,E1 -4332.687,E2 -4332.687} C_VEL
LIN {X 0,Y 532.21,Z 330.754,A -85,B 0,C 180,E1 -4333.167,E2 -4333.167} C_VEL
LIN {X 0,Y 531.734,Z 326.201,A -85,B 0,C 180,E1 -4333.302,E2 -4333.302} C_VEL
LIN {X 0,Y 530.533,Z 319.568,A -85,B 0,C 180,E1 -4333.478,E2 -4333.478} C_VEL
LIN {X 0,Y 530.547,Z 315.062,A -85,B 0,C 180,E1 -4336.152,E2 -4336.152} C_VEL
LIN {X 0,Y 530.568,Z 310.862,A -85,B 0,C 180,E1 -4338.536,E2 -4338.536} C_VEL
LIN {X 0,Y 530.646,Z 306.498,A -85,B 0,C 180,E1 -4340.953,E2 -4340.953} C_VEL
LIN {X 0,Y 530.668,Z 300.849,A -85,B 0,C 180,E1 -4343.962,E2 -4343.962} C_VEL
LIN {X 0,Y 530.6,Z 295.325,A -85,B 0,C 180,E1 -4346.766,E2 -4346.766} C_VEL
LIN {X 0,Y 530.555,Z 289.702,A -85,B 0,C 180,E1 -4349.349,E2 -4349.349} C_VEL
LIN {X 0,Y 530.564,Z 283.401,A -85,B 0,C 180,E1 -4352.031,E2 -4352.031} C_VEL
LIN {X 0,Y 530.873,Z 283.362,A -85,B 0,C 180,E1 -4353.781,E2 -4353.781} C_VEL
LIN {X 0,Y 530.955,Z 283.351,A -85,B 0,C 180,E1 -4356.559,E2 -4356.559} C_VEL
LIN {X 0,Y 530.987,Z 283.344,A -85,B 0,C 180,E1 -4359.443,E2 -4359.443} C_VEL
LIN {X 0,Y 530.967,Z 283.346,A -85,B 0,C 180,E1 -4362.458,E2 -4362.458} C_VEL
LIN {X 0,Y 530.989,Z 283.345,A -85,B 0,C 180,E1 -4365.453,E2 -4365.453} C_VEL
LIN {X 0,Y 530.991,Z 283.345,A -85,B 0,C 180,E1 -4368.564,E2 -4368.564} C_VEL
LIN {X 0,Y 531,Z 283.466,A -85,B 0,C 180,E1 -4371.342,E2 -4371.342} C_VEL
LIN {X 0,Y 532.399,Z 290.726,A -85,B 0,C 180,E1 -4373.634,E2 -4373.634} C_VEL
LIN {X 0,Y 532.578,Z 294.949,A -85,B 0,C 180,E1 -4374.902,E2 -4374.902} C_VEL
LIN {X 0,Y 532.286,Z 304.562,A -85,B 0,C 180,E1 -4377.674,E2 -4377.674} C_VEL
LIN {X 0,Y 531.99,Z 315.432,A -85,B 0,C 180,E1 -4380.738,E2 -4380.738} C_VEL
LIN {X 0,Y 531.71,Z 326.114,A -85,B 0,C 180,E1 -4383.701,E2 -4383.701} C_VEL
LIN {X 0,Y 531.496,Z 336.919,A -85,B 0,C 180,E1 -4386.628,E2 -4386.628} C_VEL
LIN {X 0,Y 531.202,Z 349.197,A -85,B 0,C 180,E1 -4389.88,E2 -4389.88} C_VEL
LIN {X 0,Y 530.985,Z 361.475,A -85,B 0,C 180,E1 -4393.071,E2 -4393.071} C_VEL
LIN {X 0,Y 530.767,Z 374.52,A -85,B 0,C 180,E1 -4396.406,E2 -4396.406} C_VEL
LIN {X 0,Y 530.756,Z 374.712,A -85,B 0,C 180,E1 -4396.455,E2 -4396.455} C_VEL
LIN {X 0,Y 532.315,Z 385.435,A -85,B 0,C 180,E1 -4396.714,E2 -4396.714} C_VEL
LIN {X 0,Y 532.149,Z 398.473,A -85,B 0,C 180,E1 -4397.123,E2 -4397.123} C_VEL
LIN {X 0,Y 531.912,Z 409.486,A -85,B 0,C 180,E1 -4397.602,E2 -4397.602} C_VEL
LIN {X 0,Y 531.682,Z 421.021,A -85,B 0,C 180,E1 -4398.254,E2 -4398.254} C_VEL
LIN {X 0,Y 531.43,Z 431.924,A -85,B 0,C 180,E1 -4399.041,E2 -4399.041} C_VEL
LIN {X 0,Y 531.192,Z 441.6,A -85,B 0,C 180,E1 -4399.904,E2 -4399.904} C_VEL
LIN {X 0,Y 530.969,Z 450.412,A -85,B 0,C 180,E1 -4400.861,E2 -4400.861} C_VEL
LIN {X 0,Y 530.779,Z 459.002,A -85,B 0,C 180,E1 -4402.008,E2 -4402.008} C_VEL
LIN {X 0,Y 530.637,Z 465.868,A -85,B 0,C 180,E1 -4403.154,E2 -4403.154} C_VEL
LIN {X 0,Y 530.611,Z 471.366,A -85,B 0,C 180,E1 -4404.299,E2 -4404.299} C_VEL
LIN {X 0,Y 530.457,Z 475.677,A -85,B 0,C 180,E1 -4405.441,E2 -4405.441} C_VEL
LIN {X 0,Y 530.516,Z 477.957,A -85,B 0,C 180,E1 -4406.202,E2 -4406.202} C_VEL
LIN {X 0,Y 530.457,Z 479.808,A -85,B 0,C 180,E1 -4406.962,E2 -4406.962} C_VEL
LIN {X 0,Y 530.411,Z 481.197,A -85,B 0,C 180,E1 -4407.722,E2 -4407.722} C_VEL
LIN {X 0,Y 530.344,Z 482.785,A -85,B 0,C 180,E1 -4409.241,E2 -4409.241} C_VEL
LIN {X 0,Y 530.342,Z 483,A -85,B 0,C 180,E1 -4410,E2 -4410} C_VEL
LIN {X 0,Y 530.361,Z 482.186,A -85,B 0,C 180,E1 -4411.519,E2 -4411.519} C_VEL
LIN {X 0,Y 530.411,Z 481.199,A -85,B 0,C 180,E1 -4412.278,E2 -4412.278} C_VEL
LIN {X 0,Y 530.457,Z 479.81,A -85,B 0,C 180,E1 -4413.038,E2 -4413.038} C_VEL
LIN {X 0,Y 530.522,Z 476.896,A -85,B 0,C 180,E1 -4414.178,E2 -4414.178} C_VEL
LIN {X 0,Y 530.524,Z 472.949,A -85,B 0,C 180,E1 -4415.321,E2 -4415.321} C_VEL
LIN {X 0,Y 530.6,Z 467.261,A -85,B 0,C 180,E1 -4416.583,E2 -4416.583} C_VEL
LIN {X 0,Y 530.758,Z 460.237,A -85,B 0,C 180,E1 -4417.801,E2 -4417.801} C_VEL
LIN {X 0,Y 530.931,Z 451.99,A -85,B 0,C 180,E1 -4418.948,E2 -4418.948} C_VEL
LIN {X 0,Y 531.113,Z 443.538,A -85,B 0,C 180,E1 -4419.906,E2 -4419.906} C_VEL
LIN {X 0,Y 531.406,Z 433.097,A -85,B 0,C 180,E1 -4420.863,E2 -4420.863} C_VEL
LIN {X 0,Y 531.641,Z 421.313,A -85,B 0,C 180,E1 -4421.728,E2 -4421.728} C_VEL
LIN {X 0,Y 531.895,Z 409.485,A -85,B 0,C 180,E1 -4422.399,E2 -4422.399} C_VEL
LIN {X 0,Y 532.173,Z 397.168,A -85,B 0,C 180,E1 -4422.925,E2 -4422.925} C_VEL
LIN {X 0,Y 532.284,Z 384.034,A -85,B 0,C 180,E1 -4423.323,E2 -4423.323} C_VEL
LIN {X 0,Y 530.756,Z 374.712,A -85,B 0,C 180,E1 -4423.545,E2 -4423.545} C_VEL
LIN {X 0,Y 530.939,Z 363.009,A -85,B 0,C 180,E1 -4426.535,E2 -4426.535} C_VEL
LIN {X 0,Y 531.139,Z 352.266,A -85,B 0,C 180,E1 -4429.317,E2 -4429.317} C_VEL
LIN {X 0,Y 531.376,Z 341.29,A -85,B 0,C 180,E1 -4432.207,E2 -4432.207} C_VEL
LIN {X 0,Y 531.564,Z 332.314,A -85,B 0,C 180,E1 -4434.612,E2 -4434.612} C_VEL
LIN {X 0,Y 531.827,Z 321.033,A -85,B 0,C 180,E1 -4437.7,E2 -4437.7} C_VEL
LIN {X 0,Y 532.122,Z 311.049,A -85,B 0,C 180,E1 -4440.487,E2 -4440.487} C_VEL
LIN {X 0,Y 532.221,Z 300.765,A -85,B 0,C 180,E1 -4443.231,E2 -4443.231} C_VEL
LIN {X 0,Y 532.406,Z 292.563,A -85,B 0,C 180,E1 -4445.508,E2 -4445.508} C_VEL
LIN {X 0,Y 531.785,Z 287.738,A -85,B 0,C 180,E1 -4446.965,E2 -4446.965} C_VEL
LIN {X 0,Y 530.965,Z 283.35,A -85,B 0,C 180,E1 -4448.41,E2 -4448.41} C_VEL
LIN {X 0,Y 530.964,Z 283.347,A -85,B 0,C 180,E1 -4451.439,E2 -4451.439} C_VEL
LIN {X 0,Y 530.97,Z 283.349,A -85,B 0,C 180,E1 -4454.549,E2 -4454.549} C_VEL
LIN {X 0,Y 530.974,Z 283.344,A -85,B 0,C 180,E1 -4457.836,E2 -4457.836} C_VEL
LIN {X 0,Y 530.991,Z 283.345,A -85,B 0,C 180,E1 -4460.557,E2 -4460.557} C_VEL
LIN {X 0,Y 530.958,Z 283.346,A -85,B 0,C 180,E1 -4463.442,E2 -4463.442} C_VEL
LIN {X 0,Y 531.002,Z 283.341,A -85,B 0,C 180,E1 -4466.494,E2 -4466.494} C_VEL
LIN {X 0,Y 530.977,Z 283.346,A -85,B 0,C 180,E1 -4469.355,E2 -4469.355} C_VEL
LIN {X 0,Y 531.016,Z 283.338,A -85,B 0,C 180,E1 -4472.468,E2 -4472.468} C_VEL
LIN {X 0,Y 530.943,Z 283.351,A -85,B 0,C 180,E1 -4474.939,E2 -4474.939} C_VEL
LIN {X 0,Y 530.739,Z 283.556,A -85,B 0,C 180,E1 -4477.417,E2 -4477.417} C_VEL
LIN {X 0,Y 530.745,Z 285.992,A -85,B 0,C 180,E1 -4480.08,E2 -4480.08} C_VEL
LIN {X 0,Y 530.625,Z 288.697,A -85,B 0,C 180,E1 -4483.059,E2 -4483.059} C_VEL
LIN {X 0,Y 530.608,Z 290.771,A -85,B 0,C 180,E1 -4485.424,E2 -4485.424} C_VEL
LIN {X 0,Y 530.529,Z 291.924,A -85,B 0,C 180,E1 -4486.632,E2 -4486.632} C_VEL
LIN {X 0,Y 532.248,Z 301.676,A -85,B 0,C 180,E1 -4486.931,E2 -4486.931} C_VEL
LIN {X 0,Y 532.026,Z 313.693,A -85,B 0,C 180,E1 -4487.362,E2 -4487.362} C_VEL
LIN {X 0,Y 531.854,Z 324.393,A -85,B 0,C 180,E1 -4487.874,E2 -4487.874} C_VEL
LIN {X 0,Y 531.644,Z 335.67,A -85,B 0,C 180,E1 -4488.563,E2 -4488.563} C_VEL
LIN {X 0,Y 531.395,Z 346.767,A -85,B 0,C 180,E1 -4489.426,E2 -4489.426} C_VEL
LIN {X 0,Y 531.166,Z 355.675,A -85,B 0,C 180,E1 -4490.288,E2 -4490.288} C_VEL
LIN {X 0,Y 530.975,Z 363.825,A -85,B 0,C 180,E1 -4491.245,E2 -4491.245} C_VEL
LIN {X 0,Y 530.823,Z 370.592,A -85,B 0,C 180,E1 -4492.2,E2 -4492.2} C_VEL
LIN {X 0,Y 530.703,Z 376.213,A -85,B 0,C 180,E1 -4493.155,E2 -4493.155} C_VEL
LIN {X 0,Y 530.647,Z 380.018,A -85,B 0,C 180,E1 -4493.918,E2 -4493.918} C_VEL
LIN {X 0,Y 530.504,Z 384.676,A -85,B 0,C 180,E1 -4495.06,E2 -4495.06} C_VEL
LIN {X 0,Y 530.516,Z 388.237,A -85,B 0,C 180,E1 -4496.202,E2 -4496.202} C_VEL
LIN {X 0,Y 530.486,Z 390.094,A -85,B 0,C 180,E1 -4496.962,E2 -4496.962} C_VEL
LIN {X 0,Y 530.412,Z 391.538,A -85,B 0,C 180,E1 -4497.722,E2 -4497.722} C_VEL
LIN {X 0,Y 530.353,Z 393.091,A -85,B 0,C 180,E1 -4499.241,E2 -4499.241} C_VEL
LIN {X 0,Y 530.352,Z 393.359,A -85,B 0,C 180,E1 -4500,E2 -4500} C_VEL
LIN {X 0,Y 530.363,Z 392.554,A -85,B 0,C 180,E1 -4501.519,E2 -4501.519} C_VEL
LIN {X 0,Y 530.412,Z 391.655,A -85,B 0,C 180,E1 -4502.278,E2 -4502.278} C_VEL
LIN {X 0,Y 530.516,Z 388.433,A -85,B 0,C 180,E1 -4503.798,E2 -4503.798} C_VEL
LIN {X 0,Y 530.485,Z 384.931,A -85,B 0,C 180,E1 -4504.94,E2 -4504.94} C_VEL
LIN {X 0,Y 530.607,Z 380.329,A -85,B 0,C 180,E1 -4506.083,E2 -4506.083} C_VEL
LIN {X 0,Y 530.696,Z 374.518,A -85,B 0,C 180,E1 -4507.228,E2 -4507.228} C_VEL
LIN {X 0,Y 530.87,Z 367.277,A -85,B 0,C 180,E1 -4508.374,E2 -4508.374} C_VEL
LIN {X 0,Y 531.059,Z 358.076,A -85,B 0,C 180,E1 -4509.522,E2 -4509.522} C_VEL
LIN {X 0,Y 531.289,Z 349.629,A -85,B 0,C 180,E1 -4510.383,E2 -4510.383} C_VEL
LIN {X 0,Y 531.495,Z 340.577,A -85,B 0,C 180,E1 -4511.151,E2 -4511.151} C_VEL
LIN {X 0,Y 531.698,Z 331.267,A -85,B 0,C 180,E1 -4511.802,E2 -4511.802} C_VEL
LIN {X 0,Y 531.912,Z 320.763,A -85,B 0,C 180,E1 -4512.398,E2 -4512.398} C_VEL
LIN {X 0,Y 532.137,Z 308.707,A -85,B 0,C 180,E1 -4512.926,E2 -4512.926} C_VEL
LIN {X 0,Y 532.089,Z 299.812,A -85,B 0,C 180,E1 -4513.219,E2 -4513.219} C_VEL
LIN {X 0,Y 530.475,Z 291.192,A -85,B 0,C 180,E1 -4513.479,E2 -4513.479} C_VEL
LIN {X 0,Y 530.473,Z 288.338,A -85,B 0,C 180,E1 -4516.154,E2 -4516.154} C_VEL
LIN {X 0,Y 530.458,Z 285.768,A -85,B 0,C 180,E1 -4518.541,E2 -4518.541} C_VEL
LIN {X 0,Y 530.518,Z 283.405,A -85,B 0,C 180,E1 -4520.958,E2 -4520.958} C_VEL
LIN {X 0,Y 530.771,Z 283.372,A -85,B 0,C 180,E1 -4523.405,E2 -4523.405} C_VEL
LIN {X 0,Y 530.977,Z 283.339,A -85,B 0,C 180,E1 -4525.899,E2 -4525.899} C_VEL
LIN {X 0,Y 530.991,Z 283.344,A -85,B 0,C 180,E1 -4528.456,E2 -4528.456} C_VEL
LIN {X 0,Y 530.957,Z 283.342,A -85,B 0,C 180,E1 -4531.079,E2 -4531.079} C_VEL
LIN {X 0,Y 530.99,Z 283.34,A -85,B 0,C 180,E1 -4533.773,E2 -4533.773} C_VEL
LIN {X 0,Y 530.958,Z 283.348,A -85,B 0,C 180,E1 -4536.558,E2 -4536.558} C_VEL
LIN {X 0,Y 530.982,Z 283.342,A -85,B 0,C 180,E1 -4539.653,E2 -4539.653} C_VEL
LIN {X 0,Y 530.311,Z 283.431,A -85,B 0,C 180,E1 -4540.286,E2 -4540.286} C_VEL
LIN {X 0,Y 527.446,Z 283.786,A -85,B 0,C 180,E1 -4541.313,E2 -4541.313} C_VEL
LIN {X 0,Y 525.031,Z 284.089,A -85,B 0,C 180,E1 -4542.141,E2 -4542.141} C_VEL
LIN {X 0,Y 524.001,Z 284.211,A -85,B 0,C 180,E1 -4542.78,E2 -4542.78} C_VEL
LIN {X 0,Y 523.921,Z 284.22,A -85,B 0,C 180,E1 -4542.996,E2 -4542.996} C_VEL
LIN {X 0,Y 523.945,Z 284.223,A -85,B 0,C 180,E1 -4545.772,E2 -4545.772} C_VEL
LIN {X 0,Y 523.943,Z 284.216,A -85,B 0,C 180,E1 -4548.908,E2 -4548.908} C_VEL
LIN {X 0,Y 523.919,Z 284.225,A -85,B 0,C 180,E1 -4551.898,E2 -4551.898} C_VEL
LIN {X 0,Y 523.875,Z 284.228,A -85,B 0,C 180,E1 -4554.919,E2 -4554.919} C_VEL
LIN {X 0,Y 523.736,Z 284.402,A -85,B 0,C 180,E1 -4556.303,E2 -4556.303} C_VEL
LIN {X 0,Y 523.66,Z 289.906,A -85,B 0,C 180,E1 -4559.336,E2 -4559.336} C_VEL
LIN {X 0,Y 523.609,Z 295.124,A -85,B 0,C 180,E1 -4562.359,E2 -4562.359} C_VEL
LIN {X 0,Y 523.583,Z 300.283,A -85,B 0,C 180,E1 -4565.411,E2 -4565.411} C_VEL
LIN {X 0,Y 523.528,Z 304.614,A -85,B 0,C 180,E1 -4567.921,E2 -4567.921} C_VEL
LIN {X 0,Y 523.503,Z 308.97,A -85,B 0,C 180,E1 -4570.389,E2 -4570.389} C_VEL
LIN {X 0,Y 523.478,Z 313.308,A -85,B 0,C 180,E1 -4572.821,E2 -4572.821} C_VEL
LIN {X 0,Y 523.512,Z 317.584,A -85,B 0,C 180,E1 -4575.222,E2 -4575.222} C_VEL
LIN {X 0,Y 523.433,Z 319.704,A -85,B 0,C 180,E1 -4576.379,E2 -4576.379} C_VEL
LIN {X 0,Y 525.397,Z 330.105,A -85,B 0,C 180,E1 -4576.684,E2 -4576.684} C_VEL
LIN {X 0,Y 525.189,Z 343.224,A -85,B 0,C 180,E1 -4577.146,E2 -4577.146} C_VEL
LIN {X 0,Y 524.928,Z 355.063,A -85,B 0,C 180,E1 -4577.726,E2 -4577.726} C_VEL
LIN {X 0,Y 524.656,Z 367.225,A -85,B 0,C 180,E1 -4578.506,E2 -4578.506} C_VEL
LIN {X 0,Y 524.407,Z 377.942,A -85,B 0,C 180,E1 -4579.381,E2 -4579.381} C_VEL
LIN {X 0,Y 524.114,Z 387.507,A -85,B 0,C 180,E1 -4580.351,E2 -4580.351} C_VEL
LIN {X 0,Y 523.88,Z 396.795,A -85,B 0,C 180,E1 -4581.514,E2 -4581.514} C_VEL
LIN {X 0,Y 523.686,Z 404.172,A -85,B 0,C 180,E1 -4582.675,E2 -4582.675} C_VEL
LIN {X 0,Y 523.562,Z 410.096,A -85,B 0,C 180,E1 -4583.835,E2 -4583.835} C_VEL
LIN {X 0,Y 523.398,Z 414.786,A -85,B 0,C 180,E1 -4584.993,E2 -4584.993} C_VEL
LIN {X 0,Y 523.444,Z 418.367,A -85,B 0,C 180,E1 -4586.151,E2 -4586.151} C_VEL
LIN {X 0,Y 523.397,Z 420.216,A -85,B 0,C 180,E1 -4586.921,E2 -4586.921} C_VEL
LIN {X 0,Y 523.335,Z 421.632,A -85,B 0,C 180,E1 -4587.691,E2 -4587.691} C_VEL
LIN {X 0,Y 523.258,Z 423.239,A -85,B 0,C 180,E1 -4589.23,E2 -4589.23} C_VEL
LIN {X 0,Y 523.26,Z 423.476,A -85,B 0,C 180,E1 -4590,E2 -4590} C_VEL
LIN {X 0,Y 523.257,Z 423.294,A -85,B 0,C 180,E1 -4590.77,E2 -4590.77} C_VEL
LIN {X 0,Y 523.335,Z 421.758,A -85,B 0,C 180,E1 -4592.309,E2 -4592.309} C_VEL
LIN {X 0,Y 523.398,Z 420.411,A -85,B 0,C 180,E1 -4593.079,E2 -4593.079} C_VEL
LIN {X 0,Y 523.442,Z 417.573,A -85,B 0,C 180,E1 -4594.235,E2 -4594.235} C_VEL
LIN {X 0,Y 523.464,Z 413.721,A -85,B 0,C 180,E1 -4595.393,E2 -4595.393} C_VEL
LIN {X 0,Y 523.582,Z 408.302,A -85,B 0,C 180,E1 -4596.636,E2 -4596.636} C_VEL
LIN {X 0,Y 523.753,Z 401.232,A -85,B 0,C 180,E1 -4597.906,E2 -4597.906} C_VEL
LIN {X 0,Y 523.953,Z 393.137,A -85,B 0,C 180,E1 -4599.068,E2 -4599.068} C_VEL
LIN {X 0,Y 524.195,Z 384.789,A -85,B 0,C 180,E1 -4600.038,E2 -4600.038} C_VEL
LIN {X 0,Y 524.489,Z 374.527,A -85,B 0,C 180,E1 -4601.008,E2 -4601.008} C_VEL
LIN {X 0,Y 524.745,Z 363.418,A -85,B 0,C 180,E1 -4601.852,E2 -4601.852} C_VEL
LIN {X 0,Y 524.987,Z 353.209,A -85,B 0,C 180,E1 -4602.466,E2 -4602.466} C_VEL
LIN {X 0,Y 525.229,Z 340.592,A -85,B 0,C 180,E1 -4603.05,E2 -4603.05} C_VEL
LIN {X 0,Y 525.254,Z 328.996,A -85,B 0,C 180,E1 -4603.443,E2 -4603.443} C_VEL
LIN {X 0,Y 523.454,Z 319.657,A -85,B 0,C 180,E1 -4603.713,E2 -4603.713} C_VEL
LIN {X 0,Y 523.467,Z 316.325,A -85,B 0,C 180,E1 -4605.576,E2 -4605.576} C_VEL
LIN {X 0,Y 523.452,Z 312.041,A -85,B 0,C 180,E1 -4607.987,E2 -4607.987} C_VEL
LIN {X 0,Y 523.503,Z 307.691,A -85,B 0,C 180,E1 -4610.429,E2 -4610.429} C_VEL
LIN {X 0,Y 523.548,Z 303.326,A -85,B 0,C 180,E1 -4612.91,E2 -4612.91} C_VEL
LIN {X 0,Y 523.602,Z 298.166,A -85,B 0,C 180,E1 -4615.933,E2 -4615.933} C_VEL
LIN {X 0,Y 523.621,Z 293.153,A -85,B 0,C 180,E1 -4618.894,E2 -4618.894} C_VEL
LIN {X 0,Y 523.676,Z 288.494,A -85,B 0,C 180,E1 -4621.561,E2 -4621.561} C_VEL
LIN {X 0,Y 523.781,Z 284.245,A -85,B 0,C 180,E1 -4623.963,E2 -4623.963} C_VEL
LIN {X 0,Y 523.901,Z 284.227,A -85,B 0,C 180,E1 -4626.401,E2 -4626.401} C_VEL
LIN {X 0,Y 523.924,Z 284.223,A -85,B 0,C 180,E1 -4629.085,E2 -4629.085} C_VEL
LIN {X 0,Y 523.954,Z 284.221,A -85,B 0,C 180,E1 -4632.119,E2 -4632.119} C_VEL
LIN {X 0,Y 523.945,Z 284.222,A -85,B 0,C 180,E1 -4635.31,E2 -4635.31} C_VEL
LIN {X 0,Y 523.959,Z 284.221,A -85,B 0,C 180,E1 -4638.69,E2 -4638.69} C_VEL
LIN {X 0,Y 523.921,Z 284.224,A -85,B 0,C 180,E1 -4641.081,E2 -4641.081} C_VEL
LIN {X 0,Y 523.897,Z 284.228,A -85,B 0,C 180,E1 -4643.825,E2 -4643.825} C_VEL
LIN {X 0,Y 523.732,Z 284.311,A -85,B 0,C 180,E1 -4646.37,E2 -4646.37} C_VEL
LIN {X 0,Y 523.669,Z 289.652,A -85,B 0,C 180,E1 -4649.337,E2 -4649.337} C_VEL
LIN {X 0,Y 523.607,Z 295.077,A -85,B 0,C 180,E1 -4652.359,E2 -4652.359} C_VEL
LIN {X 0,Y 523.593,Z 300.449,A -85,B 0,C 180,E1 -4655.411,E2 -4655.411} C_VEL
LIN {X 0,Y 523.534,Z 304.857,A -85,B 0,C 180,E1 -4657.921,E2 -4657.921} C_VEL
LIN {X 0,Y 523.526,Z 309.147,A -85,B 0,C 180,E1 -4660.39,E2 -4660.39} C_VEL
LIN {X 0,Y 523.477,Z 313.377,A -85,B 0,C 180,E1 -4662.821,E2 -4662.821} C_VEL
LIN {X 0,Y 523.512,Z 317.48,A -85,B 0,C 180,E1 -4665.222,E2 -4665.222} C_VEL
LIN {X 0,Y 523.448,Z 319.698,A -85,B 0,C 180,E1 -4666.429,E2 -4666.429} C_VEL
LIN {X 0,Y 525.301,Z 330.19,A -85,B 0,C 180,E1 -4666.73,E2 -4666.73} C_VEL
LIN {X 0,Y 525.116,Z 343.185,A -85,B 0,C 180,E1 -4667.193,E2 -4667.193} C_VEL
LIN {X 0,Y 524.826,Z 354.397,A -85,B 0,C 180,E1 -4667.741,E2 -4667.741} C_VEL
LIN {X 0,Y 524.636,Z 363.702,A -85,B 0,C 180,E1 -4668.312,E2 -4668.312} C_VEL
LIN {X 0,Y 524.45,Z 372.826,A -85,B 0,C 180,E1 -4668.991,E2 -4668.991} C_VEL
LIN {X 0,Y 524.211,Z 381.505,A -85,B 0,C 180,E1 -4669.768,E2 -4669.768} C_VEL
LIN {X 0,Y 524.048,Z 388.807,A -85,B 0,C 180,E1 -4670.544,E2 -4670.544} C_VEL
LIN {X 0,Y 523.825,Z 396.454,A -85,B 0,C 180,E1 -4671.513,E2 -4671.513} C_VEL
LIN {X 0,Y 523.69,Z 402.813,A -85,B 0,C 180,E1 -4672.481,E2 -4672.481} C_VEL
LIN {X 0,Y 523.535,Z 409.297,A -85,B 0,C 180,E1 -4673.686,E2 -4673.686} C_VEL
LIN {X 0,Y 523.397,Z 414.753,A -85,B 0,C 180,E1 -4674.993,E2 -4674.993} C_VEL
LIN {X 0,Y 523.444,Z 418.36,A -85,B 0,C 180,E1 -4676.151,E2 -4676.151} C_VEL
LIN {X 0,Y 523.397,Z 420.195,A -85,B 0,C 180,E1 -4676.921,E2 -4676.921} C_VEL
LIN {X 0,Y 523.277,Z 422.646,A -85,B 0,C 180,E1 -4678.461,E2 -4678.461} C_VEL
LIN {X 0,Y 523.259,Z 423.269,A -85,B 0,C 180,E1 -4679.23,E2 -4679.23} C_VEL
LIN {X 0,Y 523.26,Z 423.315,A -85,B 0,C 180,E1 -4680.77,E2 -4680.77} C_VEL
LIN {X 0,Y 523.279,Z 422.767,A -85,B 0,C 180,E1 -4681.539,E2 -4681.539} C_VEL
LIN {X 0,Y 523.398,Z 420.41,A -85,B 0,C 180,E1 -4683.079,E2 -4683.079} C_VEL
LIN {X 0,Y 523.442,Z 417.548,A -85,B 0,C 180,E1 -4684.235,E2 -4684.235} C_VEL
LIN {X 0,Y 523.463,Z 413.659,A -85,B 0,C 180,E1 -4685.393,E2 -4685.393} C_VEL
LIN {X 0,Y 523.534,Z 409.8,A -85,B 0,C 180,E1 -4686.313,E2 -4686.313} C_VEL
LIN {X 0,Y 523.691,Z 403.451,A -85,B 0,C 180,E1 -4687.518,E2 -4687.518} C_VEL
LIN {X 0,Y 523.825,Z 397.214,A -85,B 0,C 180,E1 -4688.487,E2 -4688.487} C_VEL
LIN {X 0,Y 524.032,Z 389.694,A -85,B 0,C 180,E1 -4689.456,E2 -4689.456} C_VEL
LIN {X 0,Y 524.226,Z 382.52,A -85,B 0,C 180,E1 -4690.232,E2 -4690.232} C_VEL
LIN {X 0,Y 524.411,Z 374.01,A -85,B 0,C 180,E1 -4691.01,E2 -4691.01} C_VEL
LIN {X 0,Y 524.639,Z 363.839,A -85,B 0,C 180,E1 -4691.776,E2 -4691.776} C_VEL
LIN {X 0,Y 524.883,Z 352.259,A -85,B 0,C 180,E1 -4692.469,E2 -4692.469} C_VEL
LIN {X 0,Y 525.143,Z 340.43,A -85,B 0,C 180,E1 -4693.003,E2 -4693.003} C_VEL
LIN {X 0,Y 525.144,Z 329.13,A -85,B 0,C 180,E1 -4693.381,E2 -4693.381} C_VEL
LIN {X 0,Y 523.489,Z 320.055,A -85,B 0,C 180,E1 -4693.662,E2 -4693.662} C_VEL
LIN {X 0,Y 523.48,Z 315.405,A -85,B 0,C 180,E1 -4696.376,E2 -4696.376} C_VEL
LIN {X 0,Y 523.524,Z 311.112,A -85,B 0,C 180,E1 -4698.795,E2 -4698.795} C_VEL
LIN {X 0,Y 523.574,Z 306.677,A -85,B 0,C 180,E1 -4701.249,E2 -4701.249} C_VEL
LIN {X 0,Y 523.59,Z 301.254,A -85,B 0,C 180,E1 -4704.112,E2 -4704.112} C_VEL
LIN {X 0,Y 523.527,Z 295.177,A -85,B 0,C 180,E1 -4707.157,E2 -4707.157} C_VEL
LIN {X 0,Y 523.458,Z 289.415,A -85,B 0,C 180,E1 -4709.786,E2 -4709.786} C_VEL
LIN {X 0,Y 523.476,Z 284.284,A -85,B 0,C 180,E1 -4711.918,E2 -4711.918} C_VEL
LIN {X 0,Y 523.88,Z 284.231,A -85,B 0,C 180,E1 -4714.294,E2 -4714.294} C_VEL
LIN {X 0,Y 523.908,Z 284.226,A -85,B 0,C 180,E1 -4717.132,E2 -4717.132} C_VEL
LIN {X 0,Y 523.94,Z 284.223,A -85,B 0,C 180,E1 -4720.13,E2 -4720.13} C_VEL
LIN {X 0,Y 523.926,Z 284.223,A -85,B 0,C 180,E1 -4722.457,E2 -4722.457} C_VEL
LIN {X 0,Y 523.957,Z 284.22,A -85,B 0,C 180,E1 -4725.309,E2 -4725.309} C_VEL
LIN {X 0,Y 523.955,Z 284.221,A -85,B 0,C 180,E1 -4728.69,E2 -4728.69} C_VEL
LIN {X 0,Y 523.989,Z 284.415,A -85,B 0,C 180,E1 -4731.071,E2 -4731.071} C_VEL
LIN {X 0,Y 525.365,Z 291.526,A -85,B 0,C 180,E1 -4733.383,E2 -4733.383} C_VEL
LIN {X 0,Y 525.674,Z 295.673,A -85,B 0,C 180,E1 -4734.641,E2 -4734.641} C_VEL
LIN {X 0,Y 525.332,Z 306.016,A -85,B 0,C 180,E1 -4737.647,E2 -4737.647} C_VEL
LIN {X 0,Y 525.062,Z 315.911,A -85,B 0,C 180,E1 -4740.463,E2 -4740.463} C_VEL
LIN {X 0,Y 524.777,Z 326.175,A -85,B 0,C 180,E1 -4743.343,E2 -4743.343} C_VEL
LIN {X 0,Y 524.521,Z 336.919,A -85,B 0,C 180,E1 -4746.299,E2 -4746.299} C_VEL
LIN {X 0,Y 524.231,Z 347.662,A -85,B 0,C 180,E1 -4749.19,E2 -4749.19} C_VEL
LIN {X 0,Y 524.005,Z 359.136,A -85,B 0,C 180,E1 -4752.225,E2 -4752.225} C_VEL
LIN {X 0,Y 523.76,Z 370.683,A -85,B 0,C 180,E1 -4755.229,E2 -4755.229} C_VEL
LIN {X 0,Y 523.727,Z 374.712,A -85,B 0,C 180,E1 -4756.27,E2 -4756.27} C_VEL
LIN {X 0,Y 525.425,Z 385.434,A -85,B 0,C 180,E1 -4756.537,E2 -4756.537} C_VEL
LIN {X 0,Y 525.229,Z 398.474,A -85,B 0,C 180,E1 -4756.95,E2 -4756.95} C_VEL
LIN {X 0,Y 524.966,Z 409.487,A -85,B 0,C 180,E1 -4757.435,E2 -4757.435} C_VEL
LIN {X 0,Y 524.715,Z 421.637,A -85,B 0,C 180,E1 -4758.137,E2 -4758.137} C_VEL
LIN {X 0,Y 524.416,Z 433.096,A -85,B 0,C 180,E1 -4758.99,E2 -4758.99} C_VEL
LIN {X 0,Y 524.095,Z 443.538,A -85,B 0,C 180,E1 -4759.96,E2 -4759.96} C_VEL
LIN {X 0,Y 523.896,Z 451.991,A -85,B 0,C 180,E1 -4760.931,E2 -4760.931} C_VEL
LIN {X 0,Y 523.688,Z 460.237,A -85,B 0,C 180,E1 -4762.093,E2 -4762.093} C_VEL
LIN {X 0,Y 523.574,Z 465.869,A -85,B 0,C 180,E1 -4763.061,E2 -4763.061} C_VEL
LIN {X 0,Y 523.544,Z 471.366,A -85,B 0,C 180,E1 -4764.222,E2 -4764.222} C_VEL
LIN {X 0,Y 523.361,Z 475.677,A -85,B 0,C 180,E1 -4765.379,E2 -4765.379} C_VEL
LIN {X 0,Y 523.443,Z 477.957,A -85,B 0,C 180,E1 -4766.151,E2 -4766.151} C_VEL
LIN {X 0,Y 523.367,Z 479.808,A -85,B 0,C 180,E1 -4766.921,E2 -4766.921} C_VEL
LIN {X 0,Y 523.335,Z 481.197,A -85,B 0,C 180,E1 -4767.691,E2 -4767.691} C_VEL
LIN {X 0,Y 523.25,Z 482.785,A -85,B 0,C 180,E1 -4769.23,E2 -4769.23} C_VEL
LIN {X 0,Y 523.246,Z 483,A -85,B 0,C 180,E1 -4770,E2 -4770} C_VEL
LIN {X 0,Y 523.275,Z 482.186,A -85,B 0,C 180,E1 -4771.539,E2 -4771.539} C_VEL
LIN {X 0,Y 523.335,Z 481.199,A -85,B 0,C 180,E1 -4772.309,E2 -4772.309} C_VEL
LIN {X 0,Y 523.367,Z 479.81,A -85,B 0,C 180,E1 -4773.079,E2 -4773.079} C_VEL
LIN {X 0,Y 523.441,Z 476.896,A -85,B 0,C 180,E1 -4774.235,E2 -4774.235} C_VEL
LIN {X 0,Y 523.464,Z 472.949,A -85,B 0,C 180,E1 -4775.393,E2 -4775.393} C_VEL
LIN {X 0,Y 523.524,Z 467.723,A -85,B 0,C 180,E1 -4776.582,E2 -4776.582} C_VEL
LIN {X 0,Y 523.665,Z 461.468,A -85,B 0,C 180,E1 -4777.713,E2 -4777.713} C_VEL
LIN {X 0,Y 523.857,Z 453.478,A -85,B 0,C 180,E1 -4778.875,E2 -4778.875} C_VEL
LIN {X 0,Y 524.085,Z 445.335,A -85,B 0,C 180,E1 -4779.845,E2 -4779.845} C_VEL
LIN {X 0,Y 524.364,Z 435.4,A -85,B 0,C 180,E1 -4780.815,E2 -4780.815} C_VEL
LIN {X 0,Y 524.629,Z 424.243,A -85,B 0,C 180,E1 -4781.685,E2 -4781.685} C_VEL
LIN {X 0,Y 524.844,Z 413.175,A -85,B 0,C 180,E1 -4782.372,E2 -4782.372} C_VEL
LIN {X 0,Y 525.137,Z 400.977,A -85,B 0,C 180,E1 -4782.954,E2 -4782.954} C_VEL
LIN {X 0,Y 525.384,Z 388.173,A -85,B 0,C 180,E1 -4783.391,E2 -4783.391} C_VEL
LIN {X 0,Y 525.105,Z 383.075,A -85,B 0,C 180,E1 -4783.53,E2 -4783.53} C_VEL
LIN {X 0,Y 523.727,Z 374.712,A -85,B 0,C 180,E1 -4783.73,E2 -4783.73} C_VEL
LIN {X 0,Y 523.915,Z 363.009,A -85,B 0,C 180,E1 -4786.763,E2 -4786.763} C_VEL
LIN {X 0,Y 524.155,Z 351.126,A -85,B 0,C 180,E1 -4789.888,E2 -4789.888} C_VEL
LIN {X 0,Y 524.417,Z 339.988,A -85,B 0,C 180,E1 -4792.87,E2 -4792.87} C_VEL
LIN {X 0,Y 524.666,Z 329.334,A -85,B 0,C 180,E1 -4795.782,E2 -4795.782} C_VEL
LIN {X 0,Y 524.972,Z 318.502,A -85,B 0,C 180,E1 -4798.813,E2 -4798.813} C_VEL
LIN {X 0,Y 525.147,Z 308.454,A -85,B 0,C 180,E1 -4801.462,E2 -4801.462} C_VEL
LIN {X 0,Y 525.357,Z 296.989,A -85,B 0,C 180,E1 -4804.649,E2 -4804.649} C_VEL
LIN {X 0,Y 525.338,Z 292.162,A -85,B 0,C 180,E1 -4806.06,E2 -4806.06} C_VEL
LIN {X 0,Y 523.93,Z 284.226,A -85,B 0,C 180,E1 -4808.693,E2 -4808.693} C_VEL
LIN {X 0,Y 523.925,Z 284.225,A -85,B 0,C 180,E1 -4811.306,E2 -4811.306} C_VEL
LIN {X 0,Y 523.94,Z 284.225,A -85,B 0,C 180,E1 -4814.689,E2 -4814.689} C_VEL
LIN {X 0,Y 523.944,Z 284.221,A -85,B 0,C 180,E1 -4817.88,E2 -4817.88} C_VEL
LIN {X 0,Y 523.924,Z 284.222,A -85,B 0,C 180,E1 -4820.915,E2 -4820.915} C_VEL
LIN {X 0,Y 523.903,Z 284.228,A -85,B 0,C 180,E1 -4823.825,E2 -4823.825} C_VEL
LIN {X 0,Y 523.944,Z 284.219,A -85,B 0,C 180,E1 -4826.636,E2 -4826.636} C_VEL
LIN {X 0,Y 523.959,Z 284.22,A -85,B 0,C 180,E1 -4829.356,E2 -4829.356} C_VEL
LIN {X 0,Y 523.98,Z 284.216,A -85,B 0,C 180,E1 -4832.281,E2 -4832.281} C_VEL
LIN {X 0,Y 523.901,Z 284.226,A -85,B 0,C 180,E1 -4834.579,E2 -4834.579} C_VEL
LIN {X 0,Y 523.714,Z 284.253,A -85,B 0,C 180,E1 -4837.097,E2 -4837.097} C_VEL
LIN {X 0,Y 523.723,Z 286.837,A -85,B 0,C 180,E1 -4839.944,E2 -4839.944} C_VEL
LIN {X 0,Y 523.626,Z 289.465,A -85,B 0,C 180,E1 -4842.826,E2 -4842.826} C_VEL
LIN {X 0,Y 523.589,Z 291.617,A -85,B 0,C 180,E1 -4845.224,E2 -4845.224} C_VEL
LIN {X 0,Y 523.553,Z 292.886,A -85,B 0,C 180,E1 -4846.481,E2 -4846.481} C_VEL
LIN {X 0,Y 525.338,Z 301.82,A -85,B 0,C 180,E1 -4846.756,E2 -4846.756} C_VEL
LIN {X 0,Y 525.122,Z 313.984,A -85,B 0,C 180,E1 -4847.193,E2 -4847.193} C_VEL
LIN {X 0,Y 524.923,Z 325.001,A -85,B 0,C 180,E1 -4847.724,E2 -4847.724} C_VEL
LIN {X 0,Y 524.715,Z 336.11,A -85,B 0,C 180,E1 -4848.41,E2 -4848.41} C_VEL
LIN {X 0,Y 524.438,Z 347.294,A -85,B 0,C 180,E1 -4849.284,E2 -4849.284} C_VEL
LIN {X 0,Y 524.197,Z 356.255,A -85,B 0,C 180,E1 -4850.157,E2 -4850.157} C_VEL
LIN {X 0,Y 523.997,Z 364.44,A -85,B 0,C 180,E1 -4851.127,E2 -4851.127} C_VEL
LIN {X 0,Y 523.833,Z 371.235,A -85,B 0,C 180,E1 -4852.096,E2 -4852.096} C_VEL
LIN {X 0,Y 523.671,Z 378.038,A -85,B 0,C 180,E1 -4853.281,E2 -4853.281} C_VEL
LIN {X 0,Y 523.513,Z 383.998,A -85,B 0,C 180,E1 -4854.608,E2 -4854.608} C_VEL
LIN {X 0,Y 523.497,Z 387.908,A -85,B 0,C 180,E1 -4855.766,E2 -4855.766} C_VEL
LIN {X 0,Y 523.429,Z 390.798,A -85,B 0,C 180,E1 -4856.921,E2 -4856.921} C_VEL
LIN {X 0,Y 523.352,Z 392.235,A -85,B 0,C 180,E1 -4857.691,E2 -4857.691} C_VEL
LIN {X 0,Y 523.289,Z 393.791,A -85,B 0,C 180,E1 -4859.231,E2 -4859.231} C_VEL
LIN {X 0,Y 523.286,Z 394.043,A -85,B 0,C 180,E1 -4860,E2 -4860} C_VEL
LIN {X 0,Y 523.298,Z 393.229,A -85,B 0,C 180,E1 -4861.539,E2 -4861.539} C_VEL
LIN {X 0,Y 523.348,Z 392.309,A -85,B 0,C 180,E1 -4862.309,E2 -4862.309} C_VEL
LIN {X 0,Y 523.476,Z 389.073,A -85,B 0,C 180,E1 -4863.849,E2 -4863.849} C_VEL
LIN {X 0,Y 523.451,Z 385.549,A -85,B 0,C 180,E1 -4865.007,E2 -4865.007} C_VEL
LIN {X 0,Y 523.557,Z 380.923,A -85,B 0,C 180,E1 -4866.165,E2 -4866.165} C_VEL
LIN {X 0,Y 523.691,Z 375.08,A -85,B 0,C 180,E1 -4867.325,E2 -4867.325} C_VEL
LIN {X 0,Y 523.912,Z 366.357,A -85,B 0,C 180,E1 -4868.68,E2 -4868.68} C_VEL
LIN {X 0,Y 524.074,Z 358.537,A -85,B 0,C 180,E1 -4869.65,E2 -4869.65} C_VEL
LIN {X 0,Y 524.322,Z 350.051,A -85,B 0,C 180,E1 -4870.523,E2 -4870.523} C_VEL
LIN {X 0,Y 524.542,Z 340.955,A -85,B 0,C 180,E1 -4871.3,E2 -4871.3} C_VEL
LIN {X 0,Y 524.765,Z 330.381,A -85,B 0,C 180,E1 -4872.04,E2 -4872.04} C_VEL
LIN {X 0,Y 525.051,Z 318.119,A -85,B 0,C 180,E1 -4872.71,E2 -4872.71} C_VEL
LIN {X 0,Y 525.257,Z 305.265,A -85,B 0,C 180,E1 -4873.222,E2 -4873.222} C_VEL
LIN {X 0,Y 525.048,Z 300.092,A -85,B 0,C 180,E1 -4873.393,E2 -4873.393} C_VEL
LIN {X 0,Y 523.422,Z 291.694,A -85,B 0,C 180,E1 -4873.664,E2 -4873.664} C_VEL
LIN {X 0,Y 523.404,Z 288.748,A -85,B 0,C 180,E1 -4876.378,E2 -4876.378} C_VEL
LIN {X 0,Y 523.403,Z 286.129,A -85,B 0,C 180,E1 -4878.8,E2 -4878.8} C_VEL
LIN {X 0,Y 523.408,Z 284.331,A -85,B 0,C 180,E1 -4880.433,E2 -4880.433} C_VEL
LIN {X 0,Y 523.681,Z 284.255,A -85,B 0,C 180,E1 -4882.904,E2 -4882.904} C_VEL
LIN {X 0,Y 523.897,Z 284.221,A -85,B 0,C 180,E1 -4885.422,E2 -4885.422} C_VEL
LIN {X 0,Y 523.967,Z 284.213,A -85,B 0,C 180,E1 -4887.999,E2 -4887.999} C_VEL
LIN {X 0,Y 523.943,Z 284.218,A -85,B 0,C 180,E1 -4890.854,E2 -4890.854} C_VEL
LIN {X 0,Y 523.962,Z 284.215,A -85,B 0,C 180,E1 -4893.734,E2 -4893.734} C_VEL
LIN {X 0,Y 523.907,Z 284.228,A -85,B 0,C 180,E1 -4896.401,E2 -4896.401} C_VEL
LIN {X 0,Y 523.924,Z 284.218,A -85,B 0,C 180,E1 -4899.085,E2 -4899.085} C_VEL
LIN {X 0,Y 523.957,Z 284.222,A -85,B 0,C 180,E1 -4902.119,E2 -4902.119} C_VEL
LIN {X 0,Y 523.921,Z 284.22,A -85,B 0,C 180,E1 -4902.996,E2 -4902.996} C_VEL
LIN {X 0,Y 523.267,Z 284.307,A -85,B 0,C 180,E1 -4903.638,E2 -4903.638} C_VEL
LIN {X 0,Y 520.422,Z 284.661,A -85,B 0,C 180,E1 -4904.679,E2 -4904.679} C_VEL
LIN {X 0,Y 518.004,Z 284.962,A -85,B 0,C 180,E1 -4905.519,E2 -4905.519} C_VEL
LIN {X 0,Y 516.958,Z 285.091,A -85,B 0,C 180,E1 -4906.166,E2 -4906.166} C_VEL
LIN {X 0,Y 516.869,Z 285.099,A -85,B 0,C 180,E1 -4906.386,E2 -4906.386} C_VEL
LIN {X 0,Y 516.886,Z 285.098,A -85,B 0,C 180,E1 -4909.258,E2 -4909.258} C_VEL
LIN {X 0,Y 516.866,Z 285.099,A -85,B 0,C 180,E1 -4912.274,E2 -4912.274} C_VEL
LIN {X 0,Y 516.836,Z 285.108,A -85,B 0,C 180,E1 -4915.171,E2 -4915.171} C_VEL
LIN {X 0,Y 516.682,Z 285.215,A -85,B 0,C 180,E1 -4916.338,E2 -4916.338} C_VEL
LIN {X 0,Y 516.602,Z 289.997,A -85,B 0,C 180,E1 -4918.99,E2 -4918.99} C_VEL
LIN {X 0,Y 516.54,Z 295.501,A -85,B 0,C 180,E1 -4922.176,E2 -4922.176} C_VEL
LIN {X 0,Y 516.537,Z 300.325,A -85,B 0,C 180,E1 -4925.052,E2 -4925.052} C_VEL
LIN {X 0,Y 516.481,Z 304.832,A -85,B 0,C 180,E1 -4927.715,E2 -4927.715} C_VEL
LIN {X 0,Y 516.397,Z 310.51,A -85,B 0,C 180,E1 -4930.935,E2 -4930.935} C_VEL
LIN {X 0,Y 516.376,Z 314.911,A -85,B 0,C 180,E1 -4933.392,E2 -4933.392} C_VEL
LIN {X 0,Y 516.39,Z 319.913,A -85,B 0,C 180,E1 -4936.171,E2 -4936.171} C_VEL
LIN {X 0,Y 518.475,Z 331.313,A -85,B 0,C 180,E1 -4936.527,E2 -4936.527} C_VEL
LIN {X 0,Y 518.299,Z 343.61,A -85,B 0,C 180,E1 -4936.972,E2 -4936.972} C_VEL
LIN {X 0,Y 518.005,Z 355.747,A -85,B 0,C 180,E1 -4937.576,E2 -4937.576} C_VEL
LIN {X 0,Y 517.719,Z 367.626,A -85,B 0,C 180,E1 -4938.35,E2 -4938.35} C_VEL
LIN {X 0,Y 517.447,Z 378.347,A -85,B 0,C 180,E1 -4939.237,E2 -4939.237} C_VEL
LIN {X 0,Y 517.13,Z 387.914,A -85,B 0,C 180,E1 -4940.219,E2 -4940.219} C_VEL
LIN {X 0,Y 516.859,Z 397.206,A -85,B 0,C 180,E1 -4941.398,E2 -4941.398} C_VEL
LIN {X 0,Y 516.649,Z 404.585,A -85,B 0,C 180,E1 -4942.575,E2 -4942.575} C_VEL
LIN {X 0,Y 516.514,Z 410.509,A -85,B 0,C 180,E1 -4943.751,E2 -4943.751} C_VEL
LIN {X 0,Y 516.331,Z 415.201,A -85,B 0,C 180,E1 -4944.924,E2 -4944.924} C_VEL
LIN {X 0,Y 516.373,Z 418.782,A -85,B 0,C 180,E1 -4946.098,E2 -4946.098} C_VEL
LIN {X 0,Y 516.339,Z 420.631,A -85,B 0,C 180,E1 -4946.879,E2 -4946.879} C_VEL
LIN {X 0,Y 516.263,Z 422.047,A -85,B 0,C 180,E1 -4947.659,E2 -4947.659} C_VEL
LIN {X 0,Y 516.171,Z 423.654,A -85,B 0,C 180,E1 -4949.22,E2 -4949.22} C_VEL
LIN {X 0,Y 516.173,Z 423.891,A -85,B 0,C 180,E1 -4950,E2 -4950} C_VEL
LIN {X 0,Y 516.17,Z 423.708,A -85,B 0,C 180,E1 -4950.78,E2 -4950.78} C_VEL
LIN {X 0,Y 516.263,Z 422.171,A -85,B 0,C 180,E1 -4952.341,E2 -4952.341} C_VEL
LIN {X 0,Y 516.34,Z 420.823,A -85,B 0,C 180,E1 -4953.121,E2 -4953.121} C_VEL
LIN {X 0,Y 516.368,Z 417.985,A -85,B 0,C 180,E1 -4954.293,E2 -4954.293} C_VEL
LIN {X 0,Y 516.405,Z 414.131,A -85,B 0,C 180,E1 -4955.467,E2 -4955.467} C_VEL
LIN {X 0,Y 516.538,Z 409.013,A -85,B 0,C 180,E1 -4956.666,E2 -4956.666} C_VEL
LIN {X 0,Y 516.717,Z 401.637,A -85,B 0,C 180,E1 -4958.014,E2 -4958.014} C_VEL
LIN {X 0,Y 516.94,Z 393.538,A -85,B 0,C 180,E1 -4959.192,E2 -4959.192} C_VEL
LIN {X 0,Y 517.229,Z 385.184,A -85,B 0,C 180,E1 -4960.174,E2 -4960.174} C_VEL
LIN {X 0,Y 517.542,Z 374.917,A -85,B 0,C 180,E1 -4961.158,E2 -4961.158} C_VEL
LIN {X 0,Y 517.805,Z 364.361,A -85,B 0,C 180,E1 -4961.975,E2 -4961.975} C_VEL
LIN {X 0,Y 518.07,Z 353.58,A -85,B 0,C 180,E1 -4962.636,E2 -4962.636} C_VEL
LIN {X 0,Y 518.327,Z 340.947,A -85,B 0,C 180,E1 -4963.227,E2 -4963.227} C_VEL
LIN {X 0,Y 518.376,Z 330.16,A -85,B 0,C 180,E1 -4963.6,E2 -4963.6} C_VEL
LIN {X 0,Y 516.404,Z 319.957,A -85,B 0,C 180,E1 -4963.904,E2 -4963.904} C_VEL
LIN {X 0,Y 516.381,Z 316.548,A -85,B 0,C 180,E1 -4965.795,E2 -4965.795} C_VEL
LIN {X 0,Y 516.385,Z 312.161,A -85,B 0,C 180,E1 -4968.242,E2 -4968.242} C_VEL
LIN {X 0,Y 516.42,Z 307.727,A -85,B 0,C 180,E1 -4970.722,E2 -4970.722} C_VEL
LIN {X 0,Y 516.5,Z 303.367,A -85,B 0,C 180,E1 -4973.241,E2 -4973.241} C_VEL
LIN {X 0,Y 516.527,Z 298.55,A -85,B 0,C 180,E1 -4976.101,E2 -4976.101} C_VEL
LIN {X 0,Y 516.542,Z 294.621,A -85,B 0,C 180,E1 -4978.438,E2 -4978.438} C_VEL
LIN {X 0,Y 516.602,Z 289.979,A -85,B 0,C 180,E1 -4981.129,E2 -4981.129} C_VEL
LIN {X 0,Y 516.696,Z 285.128,A -85,B 0,C 180,E1 -4983.895,E2 -4983.895} C_VEL
LIN {X 0,Y 516.867,Z 285.106,A -85,B 0,C 180,E1 -4985.781,E2 -4985.781} C_VEL
LIN {X 0,Y 516.884,Z 285.102,A -85,B 0,C 180,E1 -4988.716,E2 -4988.716} C_VEL
LIN {X 0,Y 516.915,Z 285.096,A -85,B 0,C 180,E1 -4991.775,E2 -4991.775} C_VEL
LIN {X 0,Y 516.898,Z 285.103,A -85,B 0,C 180,E1 -4995.007,E2 -4995.007} C_VEL
LIN {X 0,Y 516.916,Z 285.096,A -85,B 0,C 180,E1 -4998.399,E2 -4998.399} C_VEL
LIN {X 0,Y 516.884,Z 285.102,A -85,B 0,C 180,E1 -5001.284,E2 -5001.284} C_VEL
LIN {X 0,Y 516.828,Z 285.108,A -85,B 0,C 180,E1 -5004.216,E2 -5004.216} C_VEL
LIN {X 0,Y 516.675,Z 285.216,A -85,B 0,C 180,E1 -5006.454,E2 -5006.454} C_VEL
LIN {X 0,Y 516.576,Z 291.176,A -85,B 0,C 180,E1 -5009.776,E2 -5009.776} C_VEL
LIN {X 0,Y 516.55,Z 295.918,A -85,B 0,C 180,E1 -5012.445,E2 -5012.445} C_VEL
LIN {X 0,Y 516.545,Z 300.514,A -85,B 0,C 180,E1 -5015.053,E2 -5015.053} C_VEL
LIN {X 0,Y 516.481,Z 305.161,A -85,B 0,C 180,E1 -5017.715,E2 -5017.715} C_VEL
LIN {X 0,Y 516.45,Z 309.315,A -85,B 0,C 180,E1 -5020.11,E2 -5020.11} C_VEL
LIN {X 0,Y 516.411,Z 313.556,A -85,B 0,C 180,E1 -5022.578,E2 -5022.578} C_VEL
LIN {X 0,Y 516.446,Z 317.92,A -85,B 0,C 180,E1 -5025.061,E2 -5025.061} C_VEL
LIN {X 0,Y 516.371,Z 319.951,A -85,B 0,C 180,E1 -5026.246,E2 -5026.246} C_VEL
LIN {X 0,Y 518.385,Z 331.719,A -85,B 0,C 180,E1 -5026.6,E2 -5026.6} C_VEL
LIN {X 0,Y 518.088,Z 345.336,A -85,B 0,C 180,E1 -5027.116,E2 -5027.116} C_VEL
LIN {X 0,Y 517.86,Z 356.065,A -85,B 0,C 180,E1 -5027.666,E2 -5027.666} C_VEL
LIN {X 0,Y 517.642,Z 366.637,A -85,B 0,C 180,E1 -5028.348,E2 -5028.348} C_VEL
LIN {X 0,Y 517.345,Z 377.632,A -85,B 0,C 180,E1 -5029.234,E2 -5029.234} C_VEL
LIN {X 0,Y 517.074,Z 387.379,A -85,B 0,C 180,E1 -5030.218,E2 -5030.218} C_VEL
LIN {X 0,Y 516.851,Z 395.328,A -85,B 0,C 180,E1 -5031.201,E2 -5031.201} C_VEL
LIN {X 0,Y 516.68,Z 401.95,A -85,B 0,C 180,E1 -5032.182,E2 -5032.182} C_VEL
LIN {X 0,Y 516.54,Z 407.544,A -85,B 0,C 180,E1 -5033.178,E2 -5033.178} C_VEL
LIN {X 0,Y 516.485,Z 412.037,A -85,B 0,C 180,E1 -5034.142,E2 -5034.142} C_VEL
LIN {X 0,Y 516.339,Z 416.403,A -85,B 0,C 180,E1 -5035.316,E2 -5035.316} C_VEL
LIN {X 0,Y 516.373,Z 418.764,A -85,B 0,C 180,E1 -5036.098,E2 -5036.098} C_VEL
LIN {X 0,Y 516.339,Z 420.606,A -85,B 0,C 180,E1 -5036.879,E2 -5036.879} C_VEL
LIN {X 0,Y 516.194,Z 423.087,A -85,B 0,C 180,E1 -5038.44,E2 -5038.44} C_VEL
LIN {X 0,Y 516.174,Z 423.707,A -85,B 0,C 180,E1 -5039.22,E2 -5039.22} C_VEL
LIN {X 0,Y 516.175,Z 423.765,A -85,B 0,C 180,E1 -5040.78,E2 -5040.78} C_VEL
LIN {X 0,Y 516.196,Z 423.214,A -85,B 0,C 180,E1 -5041.56,E2 -5041.56} C_VEL
LIN {X 0,Y 516.34,Z 420.853,A -85,B 0,C 180,E1 -5043.121,E2 -5043.121} C_VEL
LIN {X 0,Y 516.368,Z 417.983,A -85,B 0,C 180,E1 -5044.293,E2 -5044.293} C_VEL
LIN {X 0,Y 516.405,Z 414.08,A -85,B 0,C 180,E1 -5045.467,E2 -5045.467} C_VEL
LIN {X 0,Y 516.518,Z 409.004,A -85,B 0,C 180,E1 -5046.646,E2 -5046.646} C_VEL
LIN {X 0,Y 516.66,Z 402.679,A -85,B 0,C 180,E1 -5047.818,E2 -5047.818} C_VEL
LIN {X 0,Y 516.897,Z 394.76,A -85,B 0,C 180,E1 -5048.996,E2 -5048.996} C_VEL
LIN {X 0,Y 517.138,Z 384.72,A -85,B 0,C 180,E1 -5050.176,E2 -5050.176} C_VEL
LIN {X 0,Y 517.442,Z 375.369,A -85,B 0,C 180,E1 -5051.061,E2 -5051.061} C_VEL
LIN {X 0,Y 517.663,Z 364.737,A -85,B 0,C 180,E1 -5051.883,E2 -5051.883} C_VEL
LIN {X 0,Y 517.945,Z 352.248,A -85,B 0,C 180,E1 -5052.639,E2 -5052.639} C_VEL
LIN {X 0,Y 518.227,Z 340.25,A -85,B 0,C 180,E1 -5053.18,E2 -5053.18} C_VEL
LIN {X 0,Y 518.207,Z 329.975,A -85,B 0,C 180,E1 -5053.53,E2 -5053.53} C_VEL
LIN {X 0,Y 516.461,Z 320.573,A -85,B 0,C 180,E1 -5053.827,E2 -5053.827} C_VEL
LIN {X 0,Y 516.419,Z 315.741,A -85,B 0,C 180,E1 -5056.606,E2 -5056.606} C_VEL
LIN {X 0,Y 516.464,Z 311.383,A -85,B 0,C 180,E1 -5059.062,E2 -5059.062} C_VEL
LIN {X 0,Y 516.502,Z 306.827,A -85,B 0,C 180,E1 -5061.555,E2 -5061.555} C_VEL
LIN {X 0,Y 516.511,Z 301.659,A -85,B 0,C 180,E1 -5064.265,E2 -5064.265} C_VEL
LIN {X 0,Y 516.457,Z 296.844,A -85,B 0,C 180,E1 -5066.684,E2 -5066.684} C_VEL
LIN {X 0,Y 516.434,Z 292.144,A -85,B 0,C 180,E1 -5068.889,E2 -5068.889} C_VEL
LIN {X 0,Y 516.447,Z 285.789,A -85,B 0,C 180,E1 -5071.596,E2 -5071.596} C_VEL
LIN {X 0,Y 516.435,Z 285.161,A -85,B 0,C 180,E1 -5071.941,E2 -5071.941} C_VEL
LIN {X 0,Y 516.818,Z 285.112,A -85,B 0,C 180,E1 -5073.951,E2 -5073.951} C_VEL
LIN {X 0,Y 516.878,Z 285.103,A -85,B 0,C 180,E1 -5076.746,E2 -5076.746} C_VEL
LIN {X 0,Y 516.884,Z 285.1,A -85,B 0,C 180,E1 -5079.721,E2 -5079.721} C_VEL
LIN {X 0,Y 516.909,Z 285.1,A -85,B 0,C 180,E1 -5081.776,E2 -5081.776} C_VEL
LIN {X 0,Y 516.926,Z 285.095,A -85,B 0,C 180,E1 -5085.01,E2 -5085.01} C_VEL
LIN {X 0,Y 516.912,Z 285.099,A -85,B 0,C 180,E1 -5088.399,E2 -5088.399} C_VEL
LIN {X 0,Y 516.924,Z 285.169,A -85,B 0,C 180,E1 -5090.723,E2 -5090.723} C_VEL
LIN {X 0,Y 518.472,Z 293.143,A -85,B 0,C 180,E1 -5093.385,E2 -5093.385} C_VEL
LIN {X 0,Y 518.741,Z 296.368,A -85,B 0,C 180,E1 -5094.38,E2 -5094.38} C_VEL
LIN {X 0,Y 518.391,Z 305.953,A -85,B 0,C 180,E1 -5097.199,E2 -5097.199} C_VEL
LIN {X 0,Y 518.17,Z 315.271,A -85,B 0,C 180,E1 -5099.878,E2 -5099.878} C_VEL
LIN {X 0,Y 517.809,Z 326.175,A -85,B 0,C 180,E1 -5102.955,E2 -5102.955} C_VEL
LIN {X 0,Y 517.535,Z 336.919,A -85,B 0,C 180,E1 -5105.959,E2 -5105.959} C_VEL
LIN {X 0,Y 517.252,Z 347.662,A -85,B 0,C 180,E1 -5108.896,E2 -5108.896} C_VEL
LIN {X 0,Y 516.978,Z 358.405,A -85,B 0,C 180,E1 -5111.78,E2 -5111.78} C_VEL
LIN {X 0,Y 516.756,Z 369.302,A -85,B 0,C 180,E1 -5114.661,E2 -5114.661} C_VEL
LIN {X 0,Y 516.681,Z 374.712,A -85,B 0,C 180,E1 -5116.079,E2 -5116.079} C_VEL
LIN {X 0,Y 518.478,Z 386.349,A -85,B 0,C 180,E1 -5116.378,E2 -5116.378} C_VEL
LIN {X 0,Y 518.301,Z 399.769,A -85,B 0,C 180,E1 -5116.822,E2 -5116.822} C_VEL
LIN {X 0,Y 517.995,Z 411.409,A -85,B 0,C 180,E1 -5117.363,E2 -5117.363} C_VEL
LIN {X 0,Y 517.714,Z 423.515,A -85,B 0,C 180,E1 -5118.106,E2 -5118.106} C_VEL
LIN {X 0,Y 517.399,Z 434.261,A -85,B 0,C 180,E1 -5118.938,E2 -5118.938} C_VEL
LIN {X 0,Y 517.081,Z 443.538,A -85,B 0,C 180,E1 -5119.823,E2 -5119.823} C_VEL
LIN {X 0,Y 516.868,Z 451.991,A -85,B 0,C 180,E1 -5120.807,E2 -5120.807} C_VEL
LIN {X 0,Y 516.641,Z 460.237,A -85,B 0,C 180,E1 -5121.985,E2 -5121.985} C_VEL
LIN {X 0,Y 516.48,Z 467.077,A -85,B 0,C 180,E1 -5123.201,E2 -5123.201} C_VEL
LIN {X 0,Y 516.405,Z 472.95,A -85,B 0,C 180,E1 -5124.533,E2 -5124.533} C_VEL
LIN {X 0,Y 516.344,Z 476.895,A -85,B 0,C 180,E1 -5125.707,E2 -5125.707} C_VEL
LIN {X 0,Y 516.282,Z 479.808,A -85,B 0,C 180,E1 -5126.879,E2 -5126.879} C_VEL
LIN {X 0,Y 516.261,Z 481.196,A -85,B 0,C 180,E1 -5127.659,E2 -5127.659} C_VEL
LIN {X 0,Y 516.16,Z 482.785,A -85,B 0,C 180,E1 -5129.22,E2 -5129.22} C_VEL
LIN {X 0,Y 516.154,Z 483,A -85,B 0,C 180,E1 -5130,E2 -5130} C_VEL
LIN {X 0,Y 516.192,Z 482.185,A -85,B 0,C 180,E1 -5131.56,E2 -5131.56} C_VEL
LIN {X 0,Y 516.261,Z 481.198,A -85,B 0,C 180,E1 -5132.341,E2 -5132.341} C_VEL
LIN {X 0,Y 516.282,Z 479.81,A -85,B 0,C 180,E1 -5133.121,E2 -5133.121} C_VEL
LIN {X 0,Y 516.344,Z 476.896,A -85,B 0,C 180,E1 -5134.293,E2 -5134.293} C_VEL
LIN {X 0,Y 516.405,Z 472.948,A -85,B 0,C 180,E1 -5135.467,E2 -5135.467} C_VEL
LIN {X 0,Y 516.487,Z 467.03,A -85,B 0,C 180,E1 -5136.808,E2 -5136.808} C_VEL
LIN {X 0,Y 516.641,Z 460.236,A -85,B 0,C 180,E1 -5138.015,E2 -5138.015} C_VEL
LIN {X 0,Y 516.868,Z 451.991,A -85,B 0,C 180,E1 -5139.193,E2 -5139.193} C_VEL
LIN {X 0,Y 517.081,Z 443.538,A -85,B 0,C 180,E1 -5140.177,E2 -5140.177} C_VEL
LIN {X 0,Y 517.461,Z 433.095,A -85,B 0,C 180,E1 -5141.159,E2 -5141.159} C_VEL
LIN {X 0,Y 517.697,Z 421.8,A -85,B 0,C 180,E1 -5142.015,E2 -5142.015} C_VEL
LIN {X 0,Y 517.98,Z 411.407,A -85,B 0,C 180,E1 -5142.638,E2 -5142.638} C_VEL
LIN {X 0,Y 518.267,Z 399.762,A -85,B 0,C 180,E1 -5143.179,E2 -5143.179} C_VEL
LIN {X 0,Y 518.478,Z 386.344,A -85,B 0,C 180,E1 -5143.622,E2 -5143.622} C_VEL
LIN {X 0,Y 516.691,Z 374.64,A -85,B 0,C 180,E1 -5143.94,E2 -5143.94} C_VEL
LIN {X 0,Y 516.906,Z 363.009,A -85,B 0,C 180,E1 -5146.997,E2 -5146.997} C_VEL
LIN {X 0,Y 517.14,Z 352.266,A -85,B 0,C 180,E1 -5149.862,E2 -5149.862} C_VEL
LIN {X 0,Y 517.46,Z 339.988,A -85,B 0,C 180,E1 -5153.196,E2 -5153.196} C_VEL
LIN {X 0,Y 517.758,Z 328.535,A -85,B 0,C 180,E1 -5156.378,E2 -5156.378} C_VEL
LIN {X 0,Y 517.964,Z 319.645,A -85,B 0,C 180,E1 -5158.795,E2 -5158.795} C_VEL
LIN {X 0,Y 518.14,Z 309.264,A -85,B 0,C 180,E1 -5161.571,E2 -5161.571} C_VEL
LIN {X 0,Y 518.377,Z 298.158,A -85,B 0,C 180,E1 -5164.71,E2 -5164.71} C_VEL
LIN {X 0,Y 518.37,Z 293.397,A -85,B 0,C 180,E1 -5166.141,E2 -5166.141} C_VEL
LIN {X 0,Y 517.023,Z 285.867,A -85,B 0,C 180,E1 -5168.703,E2 -5168.703} C_VEL
LIN {X 0,Y 516.868,Z 285.105,A -85,B 0,C 180,E1 -5169.028,E2 -5169.028} C_VEL
LIN {X 0,Y 516.885,Z 285.101,A -85,B 0,C 180,E1 -5171.778,E2 -5171.778} C_VEL
LIN {X 0,Y 516.897,Z 285.1,A -85,B 0,C 180,E1 -5175.007,E2 -5175.007} C_VEL
LIN {X 0,Y 516.912,Z 285.1,A -85,B 0,C 180,E1 -5178.399,E2 -5178.399} C_VEL
LIN {X 0,Y 516.884,Z 285.098,A -85,B 0,C 180,E1 -5181.284,E2 -5181.284} C_VEL
LIN {X 0,Y 516.874,Z 285.105,A -85,B 0,C 180,E1 -5184.22,E2 -5184.22} C_VEL
LIN {X 0,Y 516.898,Z 285.097,A -85,B 0,C 180,E1 -5187.053,E2 -5187.053} C_VEL
LIN {X 0,Y 516.895,Z 285.102,A -85,B 0,C 180,E1 -5189.796,E2 -5189.796} C_VEL
LIN {X 0,Y 516.929,Z 285.094,A -85,B 0,C 180,E1 -5192.467,E2 -5192.467} C_VEL
LIN {X 0,Y 516.83,Z 285.11,A -85,B 0,C 180,E1 -5195.068,E2 -5195.068} C_VEL
LIN {X 0,Y 516.718,Z 285.124,A -85,B 0,C 180,E1 -5196.769,E2 -5196.769} C_VEL
LIN {X 0,Y 516.677,Z 287.238,A -85,B 0,C 180,E1 -5199.289,E2 -5199.289} C_VEL
LIN {X 0,Y 516.611,Z 290.229,A -85,B 0,C 180,E1 -5202.585,E2 -5202.585} C_VEL
LIN {X 0,Y 516.499,Z 293.202,A -85,B 0,C 180,E1 -5205.823,E2 -5205.823} C_VEL
LIN {X 0,Y 516.493,Z 293.654,A -85,B 0,C 180,E1 -5206.312,E2 -5206.312} C_VEL
LIN {X 0,Y 518.357,Z 302.291,A -85,B 0,C 180,E1 -5206.587,E2 -5206.587} C_VEL
LIN {X 0,Y 518.232,Z 314.275,A -85,B 0,C 180,E1 -5207.02,E2 -5207.02} C_VEL
LIN {X 0,Y 517.991,Z 325.6,A -85,B 0,C 180,E1 -5207.569,E2 -5207.569} C_VEL
LIN {X 0,Y 517.788,Z 336.549,A -85,B 0,C 180,E1 -5208.253,E2 -5208.253} C_VEL
LIN {X 0,Y 517.484,Z 347.816,A -85,B 0,C 180,E1 -5209.138,E2 -5209.138} C_VEL
LIN {X 0,Y 517.237,Z 356.829,A -85,B 0,C 180,E1 -5210.024,E2 -5210.024} C_VEL
LIN {X 0,Y 517.026,Z 365.054,A -85,B 0,C 180,E1 -5211.007,E2 -5211.007} C_VEL
LIN {X 0,Y 516.827,Z 371.88,A -85,B 0,C 180,E1 -5211.988,E2 -5211.988} C_VEL
LIN {X 0,Y 516.681,Z 377.545,A -85,B 0,C 180,E1 -5212.968,E2 -5212.968} C_VEL
LIN {X 0,Y 516.605,Z 383.067,A -85,B 0,C 180,E1 -5214.144,E2 -5214.144} C_VEL
LIN {X 0,Y 516.413,Z 387.409,A -85,B 0,C 180,E1 -5215.316,E2 -5215.316} C_VEL
LIN {X 0,Y 516.373,Z 391.502,A -85,B 0,C 180,E1 -5216.879,E2 -5216.879} C_VEL
LIN {X 0,Y 516.292,Z 392.93,A -85,B 0,C 180,E1 -5217.66,E2 -5217.66} C_VEL
LIN {X 0,Y 516.224,Z 394.492,A -85,B 0,C 180,E1 -5219.22,E2 -5219.22} C_VEL
LIN {X 0,Y 516.22,Z 394.727,A -85,B 0,C 180,E1 -5220,E2 -5220} C_VEL
LIN {X 0,Y 516.233,Z 393.904,A -85,B 0,C 180,E1 -5221.56,E2 -5221.56} C_VEL
LIN {X 0,Y 516.283,Z 392.964,A -85,B 0,C 180,E1 -5222.341,E2 -5222.341} C_VEL
LIN {X 0,Y 516.366,Z 391.543,A -85,B 0,C 180,E1 -5223.121,E2 -5223.121} C_VEL
LIN {X 0,Y 516.444,Z 388.673,A -85,B 0,C 180,E1 -5224.292,E2 -5224.292} C_VEL
LIN {X 0,Y 516.437,Z 384.784,A -85,B 0,C 180,E1 -5225.466,E2 -5225.466} C_VEL
LIN {X 0,Y 516.598,Z 379.345,A -85,B 0,C 180,E1 -5226.722,E2 -5226.722} C_VEL
LIN {X 0,Y 516.764,Z 372.115,A -85,B 0,C 180,E1 -5228.013,E2 -5228.013} C_VEL
LIN {X 0,Y 516.954,Z 365.365,A -85,B 0,C 180,E1 -5228.995,E2 -5228.995} C_VEL
LIN {X 0,Y 517.158,Z 357.234,A -85,B 0,C 180,E1 -5229.978,E2 -5229.978} C_VEL
LIN {X 0,Y 517.459,Z 347.301,A -85,B 0,C 180,E1 -5230.961,E2 -5230.961} C_VEL
LIN {X 0,Y 517.766,Z 335.28,A -85,B 0,C 180,E1 -5231.901,E2 -5231.901} C_VEL
LIN {X 0,Y 517.97,Z 324.966,A -85,B 0,C 180,E1 -5232.538,E2 -5232.538} C_VEL
LIN {X 0,Y 518.224,Z 313.796,A -85,B 0,C 180,E1 -5233.08,E2 -5233.08} C_VEL
LIN {X 0,Y 518.228,Z 301.527,A -85,B 0,C 180,E1 -5233.529,E2 -5233.529} C_VEL
LIN {X 0,Y 516.34,Z 292.223,A -85,B 0,C 180,E1 -5233.83,E2 -5233.83} C_VEL
LIN {X 0,Y 516.334,Z 289.185,A -85,B 0,C 180,E1 -5236.609,E2 -5236.609} C_VEL
LIN {X 0,Y 516.329,Z 286.483,A -85,B 0,C 180,E1 -5239.067,E2 -5239.067} C_VEL
LIN {X 0,Y 516.365,Z 285.338,A -85,B 0,C 180,E1 -5240.094,E2 -5240.094} C_VEL
LIN {X 0,Y 516.609,Z 285.137,A -85,B 0,C 180,E1 -5242.391,E2 -5242.391} C_VEL
LIN {X 0,Y 516.822,Z 285.107,A -85,B 0,C 180,E1 -5244.933,E2 -5244.933} C_VEL
LIN {X 0,Y 516.927,Z 285.089,A -85,B 0,C 180,E1 -5247.533,E2 -5247.533} C_VEL
LIN {X 0,Y 516.89,Z 285.099,A -85,B 0,C 180,E1 -5250.204,E2 -5250.204} C_VEL
LIN {X 0,Y 516.898,Z 285.096,A -85,B 0,C 180,E1 -5252.947,E2 -5252.947} C_VEL
LIN {X 0,Y 516.874,Z 285.097,A -85,B 0,C 180,E1 -5255.78,E2 -5255.78} C_VEL
LIN {X 0,Y 516.884,Z 285.097,A -85,B 0,C 180,E1 -5258.716,E2 -5258.716} C_VEL
LIN {X 0,Y 516.917,Z 285.098,A -85,B 0,C 180,E1 -5261.775,E2 -5261.775} C_VEL
LIN {X 0,Y 516.926,Z 285.09,A -85,B 0,C 180,E1 -5265.01,E2 -5265.01} C_VEL
LIN {X 0,Y 516.869,Z 285.099,A -85,B 0,C 180,E1 -5266.386,E2 -5266.386} C_VEL
LIN {X 0,Y 516.197,Z 285.182,A -85,B 0,C 180,E1 -5267.037,E2 -5267.037} C_VEL
LIN {X 0,Y 513.358,Z 285.54,A -85,B 0,C 180,E1 -5268.094,E2 -5268.094} C_VEL
LIN {X 0,Y 510.957,Z 285.842,A -85,B 0,C 180,E1 -5268.945,E2 -5268.945} C_VEL
LIN {X 0,Y 509.918,Z 285.97,A -85,B 0,C 180,E1 -5269.602,E2 -5269.602} C_VEL
LIN {X 0,Y 509.829,Z 285.979,A -85,B 0,C 180,E1 -5269.825,E2 -5269.825} C_VEL
LIN {X 0,Y 509.82,Z 285.976,A -85,B 0,C 180,E1 -5272.659,E2 -5272.659} C_VEL
LIN {X 0,Y 509.745,Z 285.994,A -85,B 0,C 180,E1 -5275.578,E2 -5275.578} C_VEL
LIN {X 0,Y 509.641,Z 286.108,A -85,B 0,C 180,E1 -5276.407,E2 -5276.407} C_VEL
LIN {X 0,Y 509.506,Z 291.279,A -85,B 0,C 180,E1 -5279.311,E2 -5279.311} C_VEL
LIN {X 0,Y 509.483,Z 295.939,A -85,B 0,C 180,E1 -5282.03,E2 -5282.03} C_VEL
LIN {X 0,Y 509.468,Z 300.375,A -85,B 0,C 180,E1 -5284.682,E2 -5284.682} C_VEL
LIN {X 0,Y 509.412,Z 305.216,A -85,B 0,C 180,E1 -5287.572,E2 -5287.572} C_VEL
LIN {X 0,Y 509.318,Z 310.565,A -85,B 0,C 180,E1 -5290.66,E2 -5290.66} C_VEL
LIN {X 0,Y 509.307,Z 315.07,A -85,B 0,C 180,E1 -5293.155,E2 -5293.155} C_VEL
LIN {X 0,Y 509.341,Z 320.254,A -85,B 0,C 180,E1 -5295.992,E2 -5295.992} C_VEL
LIN {X 0,Y 511.592,Z 331.691,A -85,B 0,C 180,E1 -5296.343,E2 -5296.343} C_VEL
LIN {X 0,Y 511.416,Z 344.001,A -85,B 0,C 180,E1 -5296.793,E2 -5296.793} C_VEL
LIN {X 0,Y 511.104,Z 356.285,A -85,B 0,C 180,E1 -5297.414,E2 -5297.414} C_VEL
LIN {X 0,Y 510.797,Z 368.029,A -85,B 0,C 180,E1 -5298.19,E2 -5298.19} C_VEL
LIN {X 0,Y 510.489,Z 378.754,A -85,B 0,C 180,E1 -5299.088,E2 -5299.088} C_VEL
LIN {X 0,Y 510.157,Z 388.323,A -85,B 0,C 180,E1 -5300.084,E2 -5300.084} C_VEL
LIN {X 0,Y 509.92,Z 396.184,A -85,B 0,C 180,E1 -5301.08,E2 -5301.08} C_VEL
LIN {X 0,Y 509.647,Z 403.896,A -85,B 0,C 180,E1 -5302.273,E2 -5302.273} C_VEL
LIN {X 0,Y 509.478,Z 409.365,A -85,B 0,C 180,E1 -5303.319,E2 -5303.319} C_VEL
LIN {X 0,Y 509.35,Z 414.197,A -85,B 0,C 180,E1 -5304.457,E2 -5304.457} C_VEL
LIN {X 0,Y 509.308,Z 418.137,A -85,B 0,C 180,E1 -5305.647,E2 -5305.647} C_VEL
LIN {X 0,Y 509.283,Z 421.045,A -85,B 0,C 180,E1 -5306.836,E2 -5306.836} C_VEL
LIN {X 0,Y 509.193,Z 422.461,A -85,B 0,C 180,E1 -5307.627,E2 -5307.627} C_VEL
LIN {X 0,Y 509.084,Z 424.07,A -85,B 0,C 180,E1 -5309.209,E2 -5309.209} C_VEL
LIN {X 0,Y 509.086,Z 424.306,A -85,B 0,C 180,E1 -5310,E2 -5310} C_VEL
LIN {X 0,Y 509.083,Z 424.123,A -85,B 0,C 180,E1 -5310.791,E2 -5310.791} C_VEL
LIN {X 0,Y 509.194,Z 422.584,A -85,B 0,C 180,E1 -5312.373,E2 -5312.373} C_VEL
LIN {X 0,Y 509.283,Z 421.234,A -85,B 0,C 180,E1 -5313.164,E2 -5313.164} C_VEL
LIN {X 0,Y 509.299,Z 418.397,A -85,B 0,C 180,E1 -5314.353,E2 -5314.353} C_VEL
LIN {X 0,Y 509.349,Z 414.541,A -85,B 0,C 180,E1 -5315.543,E2 -5315.543} C_VEL
LIN {X 0,Y 509.507,Z 408.671,A -85,B 0,C 180,E1 -5316.911,E2 -5316.911} C_VEL
LIN {X 0,Y 509.704,Z 402.041,A -85,B 0,C 180,E1 -5318.125,E2 -5318.125} C_VEL
LIN {X 0,Y 509.933,Z 393.939,A -85,B 0,C 180,E1 -5319.32,E2 -5319.32} C_VEL
LIN {X 0,Y 510.266,Z 385.58,A -85,B 0,C 180,E1 -5320.315,E2 -5320.315} C_VEL
LIN {X 0,Y 510.603,Z 375.308,A -85,B 0,C 180,E1 -5321.311,E2 -5321.311} C_VEL
LIN {X 0,Y 510.868,Z 364.216,A -85,B 0,C 180,E1 -5322.177,E2 -5322.177} C_VEL
LIN {X 0,Y 511.232,Z 352.066,A -85,B 0,C 180,E1 -5322.908,E2 -5322.908} C_VEL
LIN {X 0,Y 511.49,Z 340.088,A -85,B 0,C 180,E1 -5323.458,E2 -5323.458} C_VEL
LIN {X 0,Y 511.463,Z 330.913,A -85,B 0,C 180,E1 -5323.775,E2 -5323.775} C_VEL
LIN {X 0,Y 509.367,Z 320.256,A -85,B 0,C 180,E1 -5324.1,E2 -5324.1} C_VEL
LIN {X 0,Y 509.306,Z 315.24,A -85,B 0,C 180,E1 -5326.845,E2 -5326.845} C_VEL
LIN {X 0,Y 509.317,Z 310.732,A -85,B 0,C 180,E1 -5329.34,E2 -5329.34} C_VEL
LIN {X 0,Y 509.412,Z 305.371,A -85,B 0,C 180,E1 -5332.429,E2 -5332.429} C_VEL
LIN {X 0,Y 509.468,Z 300.528,A -85,B 0,C 180,E1 -5335.318,E2 -5335.318} C_VEL
LIN {X 0,Y 509.474,Z 296.043,A -85,B 0,C 180,E1 -5338.011,E2 -5338.011} C_VEL
LIN {X 0,Y 509.542,Z 290.534,A -85,B 0,C 180,E1 -5341.223,E2 -5341.223} C_VEL
LIN {X 0,Y 509.621,Z 286.009,A -85,B 0,C 180,E1 -5343.821,E2 -5343.821} C_VEL
LIN {X 0,Y 509.82,Z 285.982,A -85,B 0,C 180,E1 -5345.577,E2 -5345.577} C_VEL
LIN {X 0,Y 509.853,Z 285.979,A -85,B 0,C 180,E1 -5348.338,E2 -5348.338} C_VEL
LIN {X 0,Y 509.858,Z 285.976,A -85,B 0,C 180,E1 -5351.426,E2 -5351.426} C_VEL
LIN {X 0,Y 509.842,Z 285.979,A -85,B 0,C 180,E1 -5354.67,E2 -5354.67} C_VEL
LIN {X 0,Y 509.836,Z 285.982,A -85,B 0,C 180,E1 -5357.51,E2 -5357.51} C_VEL
LIN {X 0,Y 509.85,Z 285.976,A -85,B 0,C 180,E1 -5360.648,E2 -5360.648} C_VEL
LIN {X 0,Y 509.8,Z 285.983,A -85,B 0,C 180,E1 -5363.645,E2 -5363.645} C_VEL
LIN {X 0,Y 509.625,Z 286.012,A -85,B 0,C 180,E1 -5366.478,E2 -5366.478} C_VEL
LIN {X 0,Y 509.512,Z 291.095,A -85,B 0,C 180,E1 -5369.312,E2 -5369.312} C_VEL
LIN {X 0,Y 509.483,Z 295.898,A -85,B 0,C 180,E1 -5372.03,E2 -5372.03} C_VEL
LIN {X 0,Y 509.474,Z 300.559,A -85,B 0,C 180,E1 -5374.682,E2 -5374.682} C_VEL
LIN {X 0,Y 509.422,Z 305.588,A -85,B 0,C 180,E1 -5377.569,E2 -5377.569} C_VEL
LIN {X 0,Y 509.422,Z 309.49,A -85,B 0,C 180,E1 -5379.824,E2 -5379.824} C_VEL
LIN {X 0,Y 509.372,Z 313.738,A -85,B 0,C 180,E1 -5382.329,E2 -5382.329} C_VEL
LIN {X 0,Y 509.358,Z 319.579,A -85,B 0,C 180,E1 -5385.619,E2 -5385.619} C_VEL
LIN {X 0,Y 509.327,Z 320.487,A -85,B 0,C 180,E1 -5386.077,E2 -5386.077} C_VEL
LIN {X 0,Y 511.439,Z 331.502,A -85,B 0,C 180,E1 -5386.414,E2 -5386.414} C_VEL
LIN {X 0,Y 511.171,Z 345.332,A -85,B 0,C 180,E1 -5386.938,E2 -5386.938} C_VEL
LIN {X 0,Y 510.893,Z 357.367,A -85,B 0,C 180,E1 -5387.567,E2 -5387.567} C_VEL
LIN {X 0,Y 510.66,Z 368.144,A -85,B 0,C 180,E1 -5388.288,E2 -5388.288} C_VEL
LIN {X 0,Y 510.306,Z 379.927,A -85,B 0,C 180,E1 -5389.285,E2 -5389.285} C_VEL
LIN {X 0,Y 510.035,Z 389.32,A -85,B 0,C 180,E1 -5390.282,E2 -5390.282} C_VEL
LIN {X 0,Y 509.805,Z 397.022,A -85,B 0,C 180,E1 -5391.278,E2 -5391.278} C_VEL
LIN {X 0,Y 509.617,Z 403.447,A -85,B 0,C 180,E1 -5392.273,E2 -5392.273} C_VEL
LIN {X 0,Y 509.416,Z 409.347,A -85,B 0,C 180,E1 -5393.378,E2 -5393.378} C_VEL
LIN {X 0,Y 509.349,Z 413.994,A -85,B 0,C 180,E1 -5394.457,E2 -5394.457} C_VEL
LIN {X 0,Y 509.302,Z 418.032,A -85,B 0,C 180,E1 -5395.647,E2 -5395.647} C_VEL
LIN {X 0,Y 509.283,Z 421.018,A -85,B 0,C 180,E1 -5396.836,E2 -5396.836} C_VEL
LIN {X 0,Y 509.115,Z 423.516,A -85,B 0,C 180,E1 -5398.418,E2 -5398.418} C_VEL
LIN {X 0,Y 509.088,Z 424.144,A -85,B 0,C 180,E1 -5399.209,E2 -5399.209} C_VEL
LIN {X 0,Y 509.09,Z 424.211,A -85,B 0,C 180,E1 -5400.791,E2 -5400.791} C_VEL
LIN {X 0,Y 509.116,Z 423.656,A -85,B 0,C 180,E1 -5401.582,E2 -5401.582} C_VEL
LIN {X 0,Y 509.283,Z 421.295,A -85,B 0,C 180,E1 -5403.164,E2 -5403.164} C_VEL
LIN {X 0,Y 509.299,Z 418.418,A -85,B 0,C 180,E1 -5404.353,E2 -5404.353} C_VEL
LIN {X 0,Y 509.349,Z 414.5,A -85,B 0,C 180,E1 -5405.543,E2 -5405.543} C_VEL
LIN {X 0,Y 509.467,Z 409.73,A -85,B 0,C 180,E1 -5406.671,E2 -5406.671} C_VEL
LIN {X 0,Y 509.634,Z 403.044,A -85,B 0,C 180,E1 -5407.927,E2 -5407.927} C_VEL
LIN {X 0,Y 509.893,Z 395.076,A -85,B 0,C 180,E1 -5409.12,E2 -5409.12} C_VEL
LIN {X 0,Y 510.113,Z 386.838,A -85,B 0,C 180,E1 -5410.117,E2 -5410.117} C_VEL
LIN {X 0,Y 510.42,Z 376.73,A -85,B 0,C 180,E1 -5411.114,E2 -5411.114} C_VEL
LIN {X 0,Y 510.67,Z 366.731,A -85,B 0,C 180,E1 -5411.914,E2 -5411.914} C_VEL
LIN {X 0,Y 510.942,Z 355.361,A -85,B 0,C 180,E1 -5412.64,E2 -5412.64} C_VEL
LIN {X 0,Y 511.234,Z 342.636,A -85,B 0,C 180,E1 -5413.262,E2 -5413.262} C_VEL
LIN {X 0,Y 511.256,Z 330.708,A -85,B 0,C 180,E1 -5413.685,E2 -5413.685} C_VEL
LIN {X 0,Y 509.384,Z 321.07,A -85,B 0,C 180,E1 -5413.998,E2 -5413.998} C_VEL
LIN {X 0,Y 509.366,Z 316.127,A -85,B 0,C 180,E1 -5416.843,E2 -5416.843} C_VEL
LIN {X 0,Y 509.399,Z 311.641,A -85,B 0,C 180,E1 -5419.337,E2 -5419.337} C_VEL
LIN {X 0,Y 509.477,Z 305.905,A -85,B 0,C 180,E1 -5422.446,E2 -5422.446} C_VEL
LIN {X 0,Y 509.44,Z 300.322,A -85,B 0,C 180,E1 -5425.319,E2 -5425.319} C_VEL
LIN {X 0,Y 509.409,Z 294.811,A -85,B 0,C 180,E1 -5427.997,E2 -5427.997} C_VEL
LIN {X 0,Y 509.33,Z 288.799,A -85,B 0,C 180,E1 -5430.7,E2 -5430.7} C_VEL
LIN {X 0,Y 509.385,Z 286.039,A -85,B 0,C 180,E1 -5431.853,E2 -5431.853} C_VEL
LIN {X 0,Y 509.809,Z 285.983,A -85,B 0,C 180,E1 -5434.417,E2 -5434.417} C_VEL
LIN {X 0,Y 509.818,Z 285.982,A -85,B 0,C 180,E1 -5437.341,E2 -5437.341} C_VEL
LIN {X 0,Y 509.84,Z 285.981,A -85,B 0,C 180,E1 -5440.382,E2 -5440.382} C_VEL
LIN {X 0,Y 509.807,Z 285.985,A -85,B 0,C 180,E1 -5443.06,E2 -5443.06} C_VEL
LIN {X 0,Y 509.833,Z 285.98,A -85,B 0,C 180,E1 -5445.792,E2 -5445.792} C_VEL
LIN {X 0,Y 509.855,Z 285.979,A -85,B 0,C 180,E1 -5448.574,E2 -5448.574} C_VEL
LIN {X 0,Y 509.865,Z 286.068,A -85,B 0,C 180,E1 -5450.412,E2 -5450.412} C_VEL
LIN {X 0,Y 511.554,Z 294.635,A -85,B 0,C 180,E1 -5453.346,E2 -5453.346} C_VEL
LIN {X 0,Y 511.755,Z 299.255,A -85,B 0,C 180,E1 -5454.775,E2 -5454.775} C_VEL
LIN {X 0,Y 511.413,Z 308.737,A -85,B 0,C 180,E1 -5457.591,E2 -5457.591} C_VEL
LIN {X 0,Y 511.106,Z 318.18,A -85,B 0,C 180,E1 -5460.329,E2 -5460.329} C_VEL
LIN {X 0,Y 510.788,Z 329.076,A -85,B 0,C 180,E1 -5463.425,E2 -5463.425} C_VEL
LIN {X 0,Y 510.481,Z 339.988,A -85,B 0,C 180,E1 -5466.468,E2 -5466.468} C_VEL
LIN {X 0,Y 510.142,Z 351.057,A -85,B 0,C 180,E1 -5469.522,E2 -5469.522} C_VEL
LIN {X 0,Y 509.93,Z 361.475,A -85,B 0,C 180,E1 -5472.349,E2 -5472.349} C_VEL
LIN {X 0,Y 509.633,Z 374.52,A -85,B 0,C 180,E1 -5475.831,E2 -5475.831} C_VEL
LIN {X 0,Y 509.641,Z 374.712,A -85,B 0,C 180,E1 -5475.882,E2 -5475.882} C_VEL
LIN {X 0,Y 511.577,Z 387.265,A -85,B 0,C 180,E1 -5476.216,E2 -5476.216} C_VEL
LIN {X 0,Y 511.392,Z 399.769,A -85,B 0,C 180,E1 -5476.641,E2 -5476.641} C_VEL
LIN {X 0,Y 511.055,Z 411.408,A -85,B 0,C 180,E1 -5477.188,E2 -5477.188} C_VEL
LIN {X 0,Y 510.786,Z 422.096,A -85,B 0,C 180,E1 -5477.842,E2 -5477.842} C_VEL
LIN {X 0,Y 510.449,Z 433.095,A -85,B 0,C 180,E1 -5478.685,E2 -5478.685} C_VEL
LIN {X 0,Y 510.07,Z 443.538,A -85,B 0,C 180,E1 -5479.681,E2 -5479.681} C_VEL
LIN {X 0,Y 509.846,Z 451.991,A -85,B 0,C 180,E1 -5480.679,E2 -5480.679} C_VEL
LIN {X 0,Y 509.585,Z 460.236,A -85,B 0,C 180,E1 -5481.873,E2 -5481.873} C_VEL
LIN {X 0,Y 509.419,Z 466.877,A -85,B 0,C 180,E1 -5483.067,E2 -5483.067} C_VEL
LIN {X 0,Y 509.344,Z 472.95,A -85,B 0,C 180,E1 -5484.457,E2 -5484.457} C_VEL
LIN {X 0,Y 509.234,Z 476.895,A -85,B 0,C 180,E1 -5485.647,E2 -5485.647} C_VEL
LIN {X 0,Y 509.2,Z 479.807,A -85,B 0,C 180,E1 -5486.835,E2 -5486.835} C_VEL
LIN {X 0,Y 509.161,Z 481.196,A -85,B 0,C 180,E1 -5487.627,E2 -5487.627} C_VEL
LIN {X 0,Y 509.073,Z 482.785,A -85,B 0,C 180,E1 -5489.209,E2 -5489.209} C_VEL
LIN {X 0,Y 509.065,Z 483,A -85,B 0,C 180,E1 -5490,E2 -5490} C_VEL
LIN {X 0,Y 509.112,Z 482.185,A -85,B 0,C 180,E1 -5491.582,E2 -5491.582} C_VEL
LIN {X 0,Y 509.161,Z 481.198,A -85,B 0,C 180,E1 -5492.373,E2 -5492.373} C_VEL
LIN {X 0,Y 509.2,Z 479.81,A -85,B 0,C 180,E1 -5493.165,E2 -5493.165} C_VEL
LIN {X 0,Y 509.234,Z 476.895,A -85,B 0,C 180,E1 -5494.353,E2 -5494.353} C_VEL
LIN {X 0,Y 509.345,Z 472.948,A -85,B 0,C 180,E1 -5495.543,E2 -5495.543} C_VEL
LIN {X 0,Y 509.41,Z 467.282,A -85,B 0,C 180,E1 -5496.853,E2 -5496.853} C_VEL
LIN {X 0,Y 509.585,Z 460.236,A -85,B 0,C 180,E1 -5498.127,E2 -5498.127} C_VEL
LIN {X 0,Y 509.846,Z 451.991,A -85,B 0,C 180,E1 -5499.321,E2 -5499.321} C_VEL
LIN {X 0,Y 510.07,Z 443.539,A -85,B 0,C 180,E1 -5500.319,E2 -5500.319} C_VEL
LIN {X 0,Y 510.487,Z 433.094,A -85,B 0,C 180,E1 -5501.314,E2 -5501.314} C_VEL
LIN {X 0,Y 510.73,Z 422.529,A -85,B 0,C 180,E1 -5502.129,E2 -5502.129} C_VEL
LIN {X 0,Y 511.046,Z 411.406,A -85,B 0,C 180,E1 -5502.812,E2 -5502.812} C_VEL
LIN {X 0,Y 511.366,Z 399.762,A -85,B 0,C 180,E1 -5503.36,E2 -5503.36} C_VEL
LIN {X 0,Y 511.539,Z 386.344,A -85,B 0,C 180,E1 -5503.811,E2 -5503.811} C_VEL
LIN {X 0,Y 509.615,Z 374.64,A -85,B 0,C 180,E1 -5504.137,E2 -5504.137} C_VEL
LIN {X 0,Y 509.881,Z 363.009,A -85,B 0,C 180,E1 -5507.238,E2 -5507.238} C_VEL
LIN {X 0,Y 510.12,Z 352.266,A -85,B 0,C 180,E1 -5510.147,E2 -5510.147} C_VEL
LIN {X 0,Y 510.44,Z 341.524,A -85,B 0,C 180,E1 -5513.104,E2 -5513.104} C_VEL
LIN {X 0,Y 510.667,Z 332.314,A -85,B 0,C 180,E1 -5515.691,E2 -5515.691} C_VEL
LIN {X 0,Y 510.947,Z 320.725,A -85,B 0,C 180,E1 -5518.778,E2 -5518.778} C_VEL
LIN {X 0,Y 511.136,Z 310.66,A -85,B 0,C 180,E1 -5521.517,E2 -5521.517} C_VEL
LIN {X 0,Y 511.419,Z 300.378,A -85,B 0,C 180,E1 -5524.459,E2 -5524.459} C_VEL
LIN {X 0,Y 511.413,Z 294.65,A -85,B 0,C 180,E1 -5526.223,E2 -5526.223} C_VEL
LIN {X 0,Y 510.062,Z 287.248,A -85,B 0,C 180,E1 -5528.824,E2 -5528.824} C_VEL
LIN {X 0,Y 509.834,Z 285.981,A -85,B 0,C 180,E1 -5529.354,E2 -5529.354} C_VEL
LIN {X 0,Y 509.803,Z 285.985,A -85,B 0,C 180,E1 -5532.493,E2 -5532.493} C_VEL
LIN {X 0,Y 509.841,Z 285.977,A -85,B 0,C 180,E1 -5535.33,E2 -5535.33} C_VEL
LIN {X 0,Y 509.855,Z 285.978,A -85,B 0,C 180,E1 -5538.574,E2 -5538.574} C_VEL
LIN {X 0,Y 509.854,Z 285.977,A -85,B 0,C 180,E1 -5541.786,E2 -5541.786} C_VEL
LIN {X 0,Y 509.833,Z 285.978,A -85,B 0,C 180,E1 -5544.622,E2 -5544.622} C_VEL
LIN {X 0,Y 509.864,Z 285.977,A -85,B 0,C 180,E1 -5547.481,E2 -5547.481} C_VEL
LIN {X 0,Y 509.862,Z 285.975,A -85,B 0,C 180,E1 -5550.274,E2 -5550.274} C_VEL
LIN {X 0,Y 509.879,Z 285.974,A -85,B 0,C 180,E1 -5552.944,E2 -5552.944} C_VEL
LIN {X 0,Y 509.78,Z 285.989,A -85,B 0,C 180,E1 -5555.569,E2 -5555.569} C_VEL
LIN {X 0,Y 509.714,Z 285.997,A -85,B 0,C 180,E1 -5556.431,E2 -5556.431} C_VEL
LIN {X 0,Y 509.666,Z 287.227,A -85,B 0,C 180,E1 -5558.142,E2 -5558.142} C_VEL
LIN {X 0,Y 509.615,Z 289.493,A -85,B 0,C 180,E1 -5560.672,E2 -5560.672} C_VEL
LIN {X 0,Y 509.528,Z 291.757,A -85,B 0,C 180,E1 -5563.163,E2 -5563.163} C_VEL
LIN {X 0,Y 509.495,Z 294.019,A -85,B 0,C 180,E1 -5565.623,E2 -5565.623} C_VEL
LIN {X 0,Y 509.468,Z 294.513,A -85,B 0,C 180,E1 -5566.145,E2 -5566.145} C_VEL
LIN {X 0,Y 511.262,Z 302.295,A -85,B 0,C 180,E1 -5566.397,E2 -5566.397} C_VEL
LIN {X 0,Y 511.433,Z 307.317,A -85,B 0,C 180,E1 -5566.566,E2 -5566.566} C_VEL
LIN {X 0,Y 511.22,Z 320.101,A -85,B 0,C 180,E1 -5567.091,E2 -5567.091} C_VEL
LIN {X 0,Y 510.974,Z 331.816,A -85,B 0,C 180,E1 -5567.745,E2 -5567.745} C_VEL
LIN {X 0,Y 510.704,Z 343.603,A -85,B 0,C 180,E1 -5568.59,E2 -5568.59} C_VEL
LIN {X 0,Y 510.403,Z 353.583,A -85,B 0,C 180,E1 -5569.488,E2 -5569.488} C_VEL
LIN {X 0,Y 510.133,Z 362.57,A -85,B 0,C 180,E1 -5570.484,E2 -5570.484} C_VEL
LIN {X 0,Y 509.868,Z 371.286,A -85,B 0,C 180,E1 -5571.678,E2 -5571.678} C_VEL
LIN {X 0,Y 509.66,Z 378.213,A -85,B 0,C 180,E1 -5572.871,E2 -5572.871} C_VEL
LIN {X 0,Y 509.583,Z 383.75,A -85,B 0,C 180,E1 -5574.063,E2 -5574.063} C_VEL
LIN {X 0,Y 509.373,Z 388.098,A -85,B 0,C 180,E1 -5575.251,E2 -5575.251} C_VEL
LIN {X 0,Y 509.403,Z 390.332,A -85,B 0,C 180,E1 -5576.044,E2 -5576.044} C_VEL
LIN {X 0,Y 509.317,Z 392.205,A -85,B 0,C 180,E1 -5576.836,E2 -5576.836} C_VEL
LIN {X 0,Y 509.232,Z 393.625,A -85,B 0,C 180,E1 -5577.627,E2 -5577.627} C_VEL
LIN {X 0,Y 509.16,Z 395.191,A -85,B 0,C 180,E1 -5579.209,E2 -5579.209} C_VEL
LIN {X 0,Y 509.154,Z 395.41,A -85,B 0,C 180,E1 -5580,E2 -5580} C_VEL
LIN {X 0,Y 509.168,Z 394.579,A -85,B 0,C 180,E1 -5581.582,E2 -5581.582} C_VEL
LIN {X 0,Y 509.22,Z 393.618,A -85,B 0,C 180,E1 -5582.373,E2 -5582.373} C_VEL
LIN {X 0,Y 509.31,Z 392.196,A -85,B 0,C 180,E1 -5583.164,E2 -5583.164} C_VEL
LIN {X 0,Y 509.405,Z 389.3,A -85,B 0,C 180,E1 -5584.352,E2 -5584.352} C_VEL
LIN {X 0,Y 509.393,Z 385.383,A -85,B 0,C 180,E1 -5585.542,E2 -5585.542} C_VEL
LIN {X 0,Y 509.583,Z 380.075,A -85,B 0,C 180,E1 -5586.781,E2 -5586.781} C_VEL
LIN {X 0,Y 509.728,Z 373.888,A -85,B 0,C 180,E1 -5587.925,E2 -5587.925} C_VEL
LIN {X 0,Y 509.933,Z 367.349,A -85,B 0,C 180,E1 -5588.92,E2 -5588.92} C_VEL
LIN {X 0,Y 510.124,Z 359.458,A -85,B 0,C 180,E1 -5589.917,E2 -5589.917} C_VEL
LIN {X 0,Y 510.466,Z 349.846,A -85,B 0,C 180,E1 -5590.912,E2 -5590.912} C_VEL
LIN {X 0,Y 510.757,Z 339.143,A -85,B 0,C 180,E1 -5591.811,E2 -5591.811} C_VEL
LIN {X 0,Y 510.957,Z 327.77,A -85,B 0,C 180,E1 -5592.569,E2 -5592.569} C_VEL
LIN {X 0,Y 511.293,Z 315.148,A -85,B 0,C 180,E1 -5593.21,E2 -5593.21} C_VEL
LIN {X 0,Y 511.417,Z 303.149,A -85,B 0,C 180,E1 -5593.662,E2 -5593.662} C_VEL
LIN {X 0,Y 509.3,Z 292.762,A -85,B 0,C 180,E1 -5594,E2 -5594} C_VEL
LIN {X 0,Y 509.265,Z 289.595,A -85,B 0,C 180,E1 -5596.846,E2 -5596.846} C_VEL
LIN {X 0,Y 509.258,Z 286.82,A -85,B 0,C 180,E1 -5599.342,E2 -5599.342} C_VEL
LIN {X 0,Y 509.309,Z 286.047,A -85,B 0,C 180,E1 -5600.225,E2 -5600.225} C_VEL
LIN {X 0,Y 509.59,Z 286.011,A -85,B 0,C 180,E1 -5602.716,E2 -5602.716} C_VEL
LIN {X 0,Y 509.794,Z 285.978,A -85,B 0,C 180,E1 -5605.301,E2 -5605.301} C_VEL
LIN {X 0,Y 509.897,Z 285.967,A -85,B 0,C 180,E1 -5608.1,E2 -5608.1} C_VEL
LIN {X 0,Y 509.848,Z 285.97,A -85,B 0,C 180,E1 -5611.28,E2 -5611.28} C_VEL
LIN {X 0,Y 509.859,Z 285.978,A -85,B 0,C 180,E1 -5614.203,E2 -5614.203} C_VEL
LIN {X 0,Y 509.82,Z 285.977,A -85,B 0,C 180,E1 -5617.341,E2 -5617.341} C_VEL
LIN {X 0,Y 509.841,Z 285.979,A -85,B 0,C 180,E1 -5620.382,E2 -5620.382} C_VEL
LIN {X 0,Y 509.827,Z 285.976,A -85,B 0,C 180,E1 -5623.062,E2 -5623.062} C_VEL
LIN {X 0,Y 509.835,Z 285.981,A -85,B 0,C 180,E1 -5625.792,E2 -5625.792} C_VEL
LIN {X 0,Y 509.859,Z 285.971,A -85,B 0,C 180,E1 -5628.575,E2 -5628.575} C_VEL
LIN {X 0,Y 509.829,Z 285.979,A -85,B 0,C 180,E1 -5629.825,E2 -5629.825} C_VEL
LIN {X 0,Y 509.152,Z 286.061,A -85,B 0,C 180,E1 -5630.485,E2 -5630.485} C_VEL
LIN {X 0,Y 506.303,Z 286.421,A -85,B 0,C 180,E1 -5631.556,E2 -5631.556} C_VEL
LIN {X 0,Y 503.894,Z 286.719,A -85,B 0,C 180,E1 -5632.419,E2 -5632.419} C_VEL
LIN {X 0,Y 502.849,Z 286.847,A -85,B 0,C 180,E1 -5633.085,E2 -5633.085} C_VEL
LIN {X 0,Y 502.757,Z 286.857,A -85,B 0,C 180,E1 -5633.311,E2 -5633.311} C_VEL
LIN {X 0,Y 502.616,Z 286.882,A -85,B 0,C 180,E1 -5636.233,E2 -5636.233} C_VEL
LIN {X 0,Y 502.585,Z 286.982,A -85,B 0,C 180,E1 -5636.471,E2 -5636.471} C_VEL
LIN {X 0,Y 502.471,Z 291.177,A -85,B 0,C 180,E1 -5638.834,E2 -5638.834} C_VEL
LIN {X 0,Y 502.426,Z 296.24,A -85,B 0,C 180,E1 -5641.794,E2 -5641.794} C_VEL
LIN {X 0,Y 502.384,Z 300.423,A -85,B 0,C 180,E1 -5644.299,E2 -5644.299} C_VEL
LIN {X 0,Y 502.349,Z 305.623,A -85,B 0,C 180,E1 -5647.423,E2 -5647.423} C_VEL
LIN {X 0,Y 502.261,Z 310.676,A -85,B 0,C 180,E1 -5650.377,E2 -5650.377} C_VEL
LIN {X 0,Y 502.243,Z 315.185,A -85,B 0,C 180,E1 -5652.911,E2 -5652.911} C_VEL
LIN {X 0,Y 502.298,Z 320.499,A -85,B 0,C 180,E1 -5655.775,E2 -5655.775} C_VEL
LIN {X 0,Y 504.704,Z 332.907,A -85,B 0,C 180,E1 -5656.178,E2 -5656.178} C_VEL
LIN {X 0,Y 504.531,Z 345.534,A -85,B 0,C 180,E1 -5656.661,E2 -5656.661} C_VEL
LIN {X 0,Y 504.139,Z 358.084,A -85,B 0,C 180,E1 -5657.322,E2 -5657.322} C_VEL
LIN {X 0,Y 503.868,Z 368.436,A -85,B 0,C 180,E1 -5658.025,E2 -5658.025} C_VEL
LIN {X 0,Y 503.539,Z 379.162,A -85,B 0,C 180,E1 -5658.936,E2 -5658.936} C_VEL
LIN {X 0,Y 503.166,Z 388.734,A -85,B 0,C 180,E1 -5659.945,E2 -5659.945} C_VEL
LIN {X 0,Y 502.909,Z 396.596,A -85,B 0,C 180,E1 -5660.955,E2 -5660.955} C_VEL
LIN {X 0,Y 502.626,Z 404.309,A -85,B 0,C 180,E1 -5662.164,E2 -5662.164} C_VEL
LIN {X 0,Y 502.439,Z 410.057,A -85,B 0,C 180,E1 -5663.283,E2 -5663.283} C_VEL
LIN {X 0,Y 502.297,Z 414.611,A -85,B 0,C 180,E1 -5664.379,E2 -5664.379} C_VEL
LIN {X 0,Y 502.244,Z 418.552,A -85,B 0,C 180,E1 -5665.586,E2 -5665.586} C_VEL
LIN {X 0,Y 502.228,Z 421.459,A -85,B 0,C 180,E1 -5666.791,E2 -5666.791} C_VEL
LIN {X 0,Y 502.127,Z 422.876,A -85,B 0,C 180,E1 -5667.593,E2 -5667.593} C_VEL
LIN {X 0,Y 502,Z 424.485,A -85,B 0,C 180,E1 -5669.198,E2 -5669.198} C_VEL
LIN {X 0,Y 502,Z 424.721,A -85,B 0,C 180,E1 -5670,E2 -5670} C_VEL
LIN {X 0,Y 502.037,Z 423.957,A -85,B 0,C 180,E1 -5671.604,E2 -5671.604} C_VEL
LIN {X 0,Y 502.228,Z 421.645,A -85,B 0,C 180,E1 -5673.209,E2 -5673.209} C_VEL
LIN {X 0,Y 502.231,Z 418.808,A -85,B 0,C 180,E1 -5674.414,E2 -5674.414} C_VEL
LIN {X 0,Y 502.296,Z 414.95,A -85,B 0,C 180,E1 -5675.621,E2 -5675.621} C_VEL
LIN {X 0,Y 502.476,Z 409.275,A -85,B 0,C 180,E1 -5676.967,E2 -5676.967} C_VEL
LIN {X 0,Y 502.672,Z 402.446,A -85,B 0,C 180,E1 -5678.239,E2 -5678.239} C_VEL
LIN {X 0,Y 502.933,Z 394.341,A -85,B 0,C 180,E1 -5679.451,E2 -5679.451} C_VEL
LIN {X 0,Y 503.305,Z 385.977,A -85,B 0,C 180,E1 -5680.459,E2 -5680.459} C_VEL
LIN {X 0,Y 503.659,Z 375.702,A -85,B 0,C 180,E1 -5681.469,E2 -5681.469} C_VEL
LIN {X 0,Y 503.956,Z 364.602,A -85,B 0,C 180,E1 -5682.346,E2 -5682.346} C_VEL
LIN {X 0,Y 504.325,Z 352.443,A -85,B 0,C 180,E1 -5683.088,E2 -5683.088} C_VEL
LIN {X 0,Y 504.62,Z 340.449,A -85,B 0,C 180,E1 -5683.644,E2 -5683.644} C_VEL
LIN {X 0,Y 504.584,Z 332.086,A -85,B 0,C 180,E1 -5683.941,E2 -5683.941} C_VEL
LIN {X 0,Y 502.295,Z 320.541,A -85,B 0,C 180,E1 -5684.303,E2 -5684.303} C_VEL
LIN {X 0,Y 502.242,Z 315.357,A -85,B 0,C 180,E1 -5687.089,E2 -5687.089} C_VEL
LIN {X 0,Y 502.26,Z 310.841,A -85,B 0,C 180,E1 -5689.623,E2 -5689.623} C_VEL
LIN {X 0,Y 502.348,Z 304.975,A -85,B 0,C 180,E1 -5693.062,E2 -5693.062} C_VEL
LIN {X 0,Y 502.38,Z 300.575,A -85,B 0,C 180,E1 -5695.701,E2 -5695.701} C_VEL
LIN {X 0,Y 502.413,Z 296.09,A -85,B 0,C 180,E1 -5698.399,E2 -5698.399} C_VEL
LIN {X 0,Y 502.497,Z 290.88,A -85,B 0,C 180,E1 -5701.443,E2 -5701.443} C_VEL
LIN {X 0,Y 502.578,Z 286.886,A -85,B 0,C 180,E1 -5703.77,E2 -5703.77} C_VEL
LIN {X 0,Y 502.768,Z 286.862,A -85,B 0,C 180,E1 -5705.952,E2 -5705.952} C_VEL
LIN {X 0,Y 502.805,Z 286.854,A -85,B 0,C 180,E1 -5708.976,E2 -5708.976} C_VEL
LIN {X 0,Y 502.798,Z 286.856,A -85,B 0,C 180,E1 -5712.139,E2 -5712.139} C_VEL
LIN {X 0,Y 502.788,Z 286.857,A -85,B 0,C 180,E1 -5715.47,E2 -5715.47} C_VEL
LIN {X 0,Y 502.823,Z 286.854,A -85,B 0,C 180,E1 -5718.934,E2 -5718.934} C_VEL
LIN {X 0,Y 502.794,Z 286.854,A -85,B 0,C 180,E1 -5722.046,E2 -5722.046} C_VEL
LIN {X 0,Y 502.701,Z 286.866,A -85,B 0,C 180,E1 -5725.026,E2 -5725.026} C_VEL
LIN {X 0,Y 502.54,Z 286.975,A -85,B 0,C 180,E1 -5726.588,E2 -5726.588} C_VEL
LIN {X 0,Y 502.442,Z 292.634,A -85,B 0,C 180,E1 -5729.764,E2 -5729.764} C_VEL
LIN {X 0,Y 502.387,Z 297.462,A -85,B 0,C 180,E1 -5732.507,E2 -5732.507} C_VEL
LIN {X 0,Y 502.402,Z 302.516,A -85,B 0,C 180,E1 -5735.405,E2 -5735.405} C_VEL
LIN {X 0,Y 502.34,Z 308.189,A -85,B 0,C 180,E1 -5738.669,E2 -5738.669} C_VEL
LIN {X 0,Y 502.266,Z 312.547,A -85,B 0,C 180,E1 -5741.226,E2 -5741.226} C_VEL
LIN {X 0,Y 502.267,Z 316.941,A -85,B 0,C 180,E1 -5743.749,E2 -5743.749} C_VEL
LIN {X 0,Y 502.291,Z 320.878,A -85,B 0,C 180,E1 -5745.894,E2 -5745.894} C_VEL
LIN {X 0,Y 504.544,Z 332.929,A -85,B 0,C 180,E1 -5746.276,E2 -5746.276} C_VEL
LIN {X 0,Y 504.221,Z 346.397,A -85,B 0,C 180,E1 -5746.806,E2 -5746.806} C_VEL
LIN {X 0,Y 503.947,Z 357.866,A -85,B 0,C 180,E1 -5747.419,E2 -5747.419} C_VEL
LIN {X 0,Y 503.683,Z 369.592,A -85,B 0,C 180,E1 -5748.225,E2 -5748.225} C_VEL
LIN {X 0,Y 503.334,Z 380.127,A -85,B 0,C 180,E1 -5749.135,E2 -5749.135} C_VEL
LIN {X 0,Y 503.026,Z 389.57,A -85,B 0,C 180,E1 -5750.145,E2 -5750.145} C_VEL
LIN {X 0,Y 502.774,Z 397.309,A -85,B 0,C 180,E1 -5751.155,E2 -5751.155} C_VEL
LIN {X 0,Y 502.58,Z 403.766,A -85,B 0,C 180,E1 -5752.164,E2 -5752.164} C_VEL
LIN {X 0,Y 502.369,Z 410.019,A -85,B 0,C 180,E1 -5753.352,E2 -5753.352} C_VEL
LIN {X 0,Y 502.295,Z 414.368,A -85,B 0,C 180,E1 -5754.379,E2 -5754.379} C_VEL
LIN {X 0,Y 502.234,Z 418.427,A -85,B 0,C 180,E1 -5755.586,E2 -5755.586} C_VEL
LIN {X 0,Y 502.228,Z 421.429,A -85,B 0,C 180,E1 -5756.791,E2 -5756.791} C_VEL
LIN {X 0,Y 502.039,Z 423.945,A -85,B 0,C 180,E1 -5758.396,E2 -5758.396} C_VEL
LIN {X 0,Y 502.004,Z 424.581,A -85,B 0,C 180,E1 -5759.198,E2 -5759.198} C_VEL
LIN {X 0,Y 502.006,Z 424.657,A -85,B 0,C 180,E1 -5760.802,E2 -5760.802} C_VEL
LIN {X 0,Y 502.04,Z 424.097,A -85,B 0,C 180,E1 -5761.604,E2 -5761.604} C_VEL
LIN {X 0,Y 502.228,Z 421.736,A -85,B 0,C 180,E1 -5763.209,E2 -5763.209} C_VEL
LIN {X 0,Y 502.234,Z 418.852,A -85,B 0,C 180,E1 -5764.414,E2 -5764.414} C_VEL
LIN {X 0,Y 502.295,Z 414.921,A -85,B 0,C 180,E1 -5765.621,E2 -5765.621} C_VEL
LIN {X 0,Y 502.468,Z 409.197,A -85,B 0,C 180,E1 -5766.96,E2 -5766.96} C_VEL
LIN {X 0,Y 502.635,Z 402.217,A -85,B 0,C 180,E1 -5768.24,E2 -5768.24} C_VEL
LIN {X 0,Y 502.904,Z 393.83,A -85,B 0,C 180,E1 -5769.451,E2 -5769.451} C_VEL
LIN {X 0,Y 503.16,Z 385.238,A -85,B 0,C 180,E1 -5770.462,E2 -5770.462} C_VEL
LIN {X 0,Y 503.49,Z 375.788,A -85,B 0,C 180,E1 -5771.371,E2 -5771.371} C_VEL
LIN {X 0,Y 503.777,Z 364.406,A -85,B 0,C 180,E1 -5772.253,E2 -5772.253} C_VEL
LIN {X 0,Y 504.094,Z 352.17,A -85,B 0,C 180,E1 -5772.992,E2 -5772.992} C_VEL
LIN {X 0,Y 504.383,Z 339.89,A -85,B 0,C 180,E1 -5773.548,E2 -5773.548} C_VEL
LIN {X 0,Y 504.304,Z 331.448,A -85,B 0,C 180,E1 -5773.846,E2 -5773.846} C_VEL
LIN {X 0,Y 502.345,Z 321.571,A -85,B 0,C 180,E1 -5774.172,E2 -5774.172} C_VEL
LIN {X 0,Y 502.317,Z 316.456,A -85,B 0,C 180,E1 -5777.086,E2 -5777.086} C_VEL
LIN {X 0,Y 502.346,Z 311.924,A -85,B 0,C 180,E1 -5779.619,E2 -5779.619} C_VEL
LIN {X 0,Y 502.427,Z 306.404,A -85,B 0,C 180,E1 -5782.599,E2 -5782.599} C_VEL
LIN {X 0,Y 502.366,Z 300.334,A -85,B 0,C 180,E1 -5785.702,E2 -5785.702} C_VEL
LIN {X 0,Y 502.334,Z 293.739,A -85,B 0,C 180,E1 -5788.861,E2 -5788.861} C_VEL
LIN {X 0,Y 502.307,Z 287.779,A -85,B 0,C 180,E1 -5791.408,E2 -5791.408} C_VEL
LIN {X 0,Y 502.342,Z 286.916,A -85,B 0,C 180,E1 -5791.821,E2 -5791.821} C_VEL
LIN {X 0,Y 502.763,Z 286.861,A -85,B 0,C 180,E1 -5794.437,E2 -5794.437} C_VEL
LIN {X 0,Y 502.779,Z 286.858,A -85,B 0,C 180,E1 -5797.178,E2 -5797.178} C_VEL
LIN {X 0,Y 502.79,Z 286.857,A -85,B 0,C 180,E1 -5800.015,E2 -5800.015} C_VEL
LIN {X 0,Y 502.805,Z 286.854,A -85,B 0,C 180,E1 -5802.199,E2 -5802.199} C_VEL
LIN {X 0,Y 502.803,Z 286.855,A -85,B 0,C 180,E1 -5805.468,E2 -5805.468} C_VEL
LIN {X 0,Y 502.797,Z 286.856,A -85,B 0,C 180,E1 -5807.86,E2 -5807.86} C_VEL
LIN {X 0,Y 502.815,Z 286.897,A -85,B 0,C 180,E1 -5810.068,E2 -5810.068} C_VEL
LIN {X 0,Y 504.545,Z 295.82,A -85,B 0,C 180,E1 -5813.204,E2 -5813.204} C_VEL
LIN {X 0,Y 504.88,Z 299.01,A -85,B 0,C 180,E1 -5814.222,E2 -5814.222} C_VEL
LIN {X 0,Y 504.531,Z 307.187,A -85,B 0,C 180,E1 -5816.698,E2 -5816.698} C_VEL
LIN {X 0,Y 504.213,Z 317.64,A -85,B 0,C 180,E1 -5819.791,E2 -5819.791} C_VEL
LIN {X 0,Y 503.808,Z 328.571,A -85,B 0,C 180,E1 -5822.957,E2 -5822.957} C_VEL
LIN {X 0,Y 503.527,Z 339.988,A -85,B 0,C 180,E1 -5826.123,E2 -5826.123} C_VEL
LIN {X 0,Y 503.131,Z 351.592,A -85,B 0,C 180,E1 -5829.373,E2 -5829.373} C_VEL
LIN {X 0,Y 502.875,Z 363.009,A -85,B 0,C 180,E1 -5832.514,E2 -5832.514} C_VEL
LIN {X 0,Y 502.568,Z 374.712,A -85,B 0,C 180,E1 -5835.68,E2 -5835.68} C_VEL
LIN {X 0,Y 504.664,Z 387.264,A -85,B 0,C 180,E1 -5836.023,E2 -5836.023} C_VEL
LIN {X 0,Y 504.472,Z 399.77,A -85,B 0,C 180,E1 -5836.454,E2 -5836.454} C_VEL
LIN {X 0,Y 504.117,Z 411.408,A -85,B 0,C 180,E1 -5837.009,E2 -5837.009} C_VEL
LIN {X 0,Y 503.8,Z 422.997,A -85,B 0,C 180,E1 -5837.735,E2 -5837.735} C_VEL
LIN {X 0,Y 503.443,Z 434.262,A -85,B 0,C 180,E1 -5838.628,E2 -5838.628} C_VEL
LIN {X 0,Y 503.064,Z 443.538,A -85,B 0,C 180,E1 -5839.536,E2 -5839.536} C_VEL
LIN {X 0,Y 502.811,Z 451.992,A -85,B 0,C 180,E1 -5840.547,E2 -5840.547} C_VEL
LIN {X 0,Y 502.542,Z 460.236,A -85,B 0,C 180,E1 -5841.758,E2 -5841.758} C_VEL
LIN {X 0,Y 502.345,Z 466.876,A -85,B 0,C 180,E1 -5842.969,E2 -5842.969} C_VEL
LIN {X 0,Y 502.26,Z 472.95,A -85,B 0,C 180,E1 -5844.379,E2 -5844.379} C_VEL
LIN {X 0,Y 502.128,Z 476.895,A -85,B 0,C 180,E1 -5845.585,E2 -5845.585} C_VEL
LIN {X 0,Y 502.121,Z 479.807,A -85,B 0,C 180,E1 -5846.791,E2 -5846.791} C_VEL
LIN {X 0,Y 502.066,Z 481.195,A -85,B 0,C 180,E1 -5847.593,E2 -5847.593} C_VEL
LIN {X 0,Y 501.99,Z 482.786,A -85,B 0,C 180,E1 -5849.198,E2 -5849.198} C_VEL
LIN {X 0,Y 501.98,Z 483,A -85,B 0,C 180,E1 -5850,E2 -5850} C_VEL
LIN {X 0,Y 502.036,Z 482.185,A -85,B 0,C 180,E1 -5851.604,E2 -5851.604} C_VEL
LIN {X 0,Y 502.066,Z 481.197,A -85,B 0,C 180,E1 -5852.407,E2 -5852.407} C_VEL
LIN {X 0,Y 502.121,Z 479.81,A -85,B 0,C 180,E1 -5853.209,E2 -5853.209} C_VEL
LIN {X 0,Y 502.128,Z 476.895,A -85,B 0,C 180,E1 -5854.415,E2 -5854.415} C_VEL
LIN {X 0,Y 502.26,Z 472.948,A -85,B 0,C 180,E1 -5855.621,E2 -5855.621} C_VEL
LIN {X 0,Y 502.336,Z 466.976,A -85,B 0,C 180,E1 -5857.012,E2 -5857.012} C_VEL
LIN {X 0,Y 502.542,Z 460.236,A -85,B 0,C 180,E1 -5858.242,E2 -5858.242} C_VEL
LIN {X 0,Y 502.811,Z 451.991,A -85,B 0,C 180,E1 -5859.453,E2 -5859.453} C_VEL
LIN {X 0,Y 503.064,Z 443.539,A -85,B 0,C 180,E1 -5860.464,E2 -5860.464} C_VEL
LIN {X 0,Y 503.514,Z 433.094,A -85,B 0,C 180,E1 -5861.473,E2 -5861.473} C_VEL
LIN {X 0,Y 503.793,Z 421.427,A -85,B 0,C 180,E1 -5862.378,E2 -5862.378} C_VEL
LIN {X 0,Y 504.135,Z 409.488,A -85,B 0,C 180,E1 -5863.093,E2 -5863.093} C_VEL
LIN {X 0,Y 504.522,Z 397.165,A -85,B 0,C 180,E1 -5863.647,E2 -5863.647} C_VEL
LIN {X 0,Y 504.558,Z 386.8,A -85,B 0,C 180,E1 -5863.993,E2 -5863.993} C_VEL
LIN {X 0,Y 502.573,Z 374.64,A -85,B 0,C 180,E1 -5864.34,E2 -5864.34} C_VEL
LIN {X 0,Y 502.875,Z 363.009,A -85,B 0,C 180,E1 -5867.486,E2 -5867.486} C_VEL
LIN {X 0,Y 503.131,Z 351.592,A -85,B 0,C 180,E1 -5870.627,E2 -5870.627} C_VEL
LIN {X 0,Y 503.527,Z 339.988,A -85,B 0,C 180,E1 -5873.877,E2 -5873.877} C_VEL
LIN {X 0,Y 503.741,Z 328.127,A -85,B 0,C 180,E1 -5877.045,E2 -5877.045} C_VEL
LIN {X 0,Y 503.985,Z 318.445,A -85,B 0,C 180,E1 -5879.673,E2 -5879.673} C_VEL
LIN {X 0,Y 504.198,Z 308.57,A -85,B 0,C 180,E1 -5882.456,E2 -5882.456} C_VEL
LIN {X 0,Y 504.437,Z 300.546,A -85,B 0,C 180,E1 -5884.836,E2 -5884.836} C_VEL
LIN {X 0,Y 504.398,Z 295.616,A -85,B 0,C 180,E1 -5886.413,E2 -5886.413} C_VEL
LIN {X 0,Y 503.136,Z 288.648,A -85,B 0,C 180,E1 -5888.945,E2 -5888.945} C_VEL
LIN {X 0,Y 502.775,Z 286.86,A -85,B 0,C 180,E1 -5889.752,E2 -5889.752} C_VEL
LIN {X 0,Y 502.773,Z 286.861,A -85,B 0,C 180,E1 -5892.195,E2 -5892.195} C_VEL
LIN {X 0,Y 502.788,Z 286.856,A -85,B 0,C 180,E1 -5895.47,E2 -5895.47} C_VEL
LIN {X 0,Y 502.797,Z 286.855,A -85,B 0,C 180,E1 -5897.861,E2 -5897.861} C_VEL
LIN {X 0,Y 502.805,Z 286.853,A -85,B 0,C 180,E1 -5901.024,E2 -5901.024} C_VEL
